LIN {X 0,Y 418.316,Z 278.186,A -85,B 0,C 180,E1 -10001.631,E2 -10001.631} C_VEL
LIN {X 0,Y 418.304,Z 278.193,A -85,B 0,C 180,E1 -10004.596,E2 -10004.596} C_VEL
LIN {X 0,Y 418.281,Z 278.19,A -85,B 0,C 180,E1 -10007.604,E2 -10007.604} C_VEL
LIN {X 0,Y 418.25,Z 278.202,A -85,B 0,C 180,E1 -10010.662,E2 -10010.662} C_VEL
LIN {X 0,Y 418.276,Z 278.19,A -85,B 0,C 180,E1 -10013.781,E2 -10013.781} C_VEL
LIN {X 0,Y 418.309,Z 278.192,A -85,B 0,C 180,E1 -10017.07,E2 -10017.07} C_VEL
LIN {X 0,Y 418.242,Z 278.195,A -85,B 0,C 180,E1 -10020.271,E2 -10020.271} C_VEL
LIN {X 0,Y 418.244,Z 278.196,A -85,B 0,C 180,E1 -10023.676,E2 -10023.676} C_VEL
LIN {X 0,Y 418.236,Z 278.204,A -85,B 0,C 180,E1 -10027.223,E2 -10027.223} C_VEL
LIN {X 0,Y 418.247,Z 278.197,A -85,B 0,C 180,E1 -10029.681,E2 -10029.681} C_VEL
LIN {X 0,Y 418.224,Z 278.197,A -85,B 0,C 180,E1 -10032.32,E2 -10032.32} C_VEL
LIN {X 0,Y 418.253,Z 278.196,A -85,B 0,C 180,E1 -10035.111,E2 -10035.111} C_VEL
LIN {X 0,Y 418.286,Z 278.195,A -85,B 0,C 180,E1 -10037.772,E2 -10037.772} C_VEL
LIN {X 0,Y 418.258,Z 278.198,A -85,B 0,C 180,E1 -10041.559,E2 -10041.559} C_VEL
LIN {X 0,Y 418.252,Z 278.194,A -85,B 0,C 180,E1 -10045.158,E2 -10045.158} C_VEL
LIN {X 0,Y 418.237,Z 278.197,A -85,B 0,C 180,E1 -10047.471,E2 -10047.471} C_VEL
LIN {X 0,Y 418.268,Z 278.192,A -85,B 0,C 180,E1 -10050.893,E2 -10050.893} C_VEL
LIN {X 0,Y 418.262,Z 278.199,A -85,B 0,C 180,E1 -10054.095,E2 -10054.095} C_VEL
LIN {X 0,Y 418.228,Z 278.196,A -85,B 0,C 180,E1 -10057.263,E2 -10057.263} C_VEL
LIN {X 0,Y 418.272,Z 278.198,A -85,B 0,C 180,E1 -10060.364,E2 -10060.364} C_VEL
LIN {X 0,Y 418.306,Z 278.187,A -85,B 0,C 180,E1 -10063.404,E2 -10063.404} C_VEL
LIN {X 0,Y 418.335,Z 278.186,A -85,B 0,C 180,E1 -10066.999,E2 -10066.999} C_VEL
LIN {X 0,Y 418.329,Z 278.186,A -85,B 0,C 180,E1 -10070.328,E2 -10070.328} C_VEL
LIN {X 0,Y 418.479,Z 278.168,A -85,B 0,C 180,E1 -10073.249,E2 -10073.249} C_VEL
LIN {X 0,Y 418.326,Z 278.189,A -85,B 0,C 180,E1 -10075.181,E2 -10075.181} C_VEL
LIN {X 0,Y 418.532,Z 278.158,A -85,B 0,C 180,E1 -10078.075,E2 -10078.075} C_VEL
LIN {X 0,Y 418.659,Z 278.143,A -85,B 0,C 180,E1 -10080,E2 -10080} C_VEL
LIN {X 0,Y 418.489,Z 278.168,A -85,B 0,C 180,E1 -10082.888,E2 -10082.888} C_VEL
LIN {X 0,Y 418.478,Z 278.166,A -85,B 0,C 180,E1 -10086.751,E2 -10086.751} C_VEL
LIN {X 0,Y 418.333,Z 278.188,A -85,B 0,C 180,E1 -10089.671,E2 -10089.671} C_VEL
LIN {X 0,Y 418.344,Z 278.183,A -85,B 0,C 180,E1 -10093.006,E2 -10093.006} C_VEL
LIN {X 0,Y 418.301,Z 278.187,A -85,B 0,C 180,E1 -10096.736,E2 -10096.736} C_VEL
LIN {X 0,Y 418.259,Z 278.201,A -85,B 0,C 180,E1 -10099.79,E2 -10099.79} C_VEL
LIN {X 0,Y 418.221,Z 278.197,A -85,B 0,C 180,E1 -10102.737,E2 -10102.737} C_VEL
LIN {X 0,Y 418.26,Z 278.199,A -85,B 0,C 180,E1 -10105.905,E2 -10105.905} C_VEL
LIN {X 0,Y 418.255,Z 278.193,A -85,B 0,C 180,E1 -10109.163,E2 -10109.163} C_VEL
LIN {X 0,Y 418.248,Z 278.195,A -85,B 0,C 180,E1 -10112.844,E2 -10112.844} C_VEL
LIN {X 0,Y 418.236,Z 278.201,A -85,B 0,C 180,E1 -10116.239,E2 -10116.239} C_VEL
LIN {X 0,Y 418.234,Z 278.196,A -85,B 0,C 180,E1 -10119.684,E2 -10119.684} C_VEL
LIN {X 0,Y 418.221,Z 278.201,A -85,B 0,C 180,E1 -10122.322,E2 -10122.322} C_VEL
LIN {X 0,Y 418.228,Z 278.199,A -85,B 0,C 180,E1 -10125.109,E2 -10125.109} C_VEL
LIN {X 0,Y 418.227,Z 278.196,A -85,B 0,C 180,E1 -10127.767,E2 -10127.767} C_VEL
LIN {X 0,Y 418.239,Z 278.199,A -85,B 0,C 180,E1 -10130.622,E2 -10130.622} C_VEL
LIN {X 0,Y 418.237,Z 278.195,A -85,B 0,C 180,E1 -10133.976,E2 -10133.976} C_VEL
LIN {X 0,Y 418.253,Z 278.201,A -85,B 0,C 180,E1 -10137.157,E2 -10137.157} C_VEL
LIN {X 0,Y 418.257,Z 278.195,A -85,B 0,C 180,E1 -10140.838,E2 -10140.838} C_VEL
LIN {X 0,Y 418.232,Z 278.2,A -85,B 0,C 180,E1 -10144.094,E2 -10144.094} C_VEL
LIN {X 0,Y 418.297,Z 278.248,A -85,B 0,C 180,E1 -10145.383,E2 -10145.383} C_VEL
LIN {X 0,Y 419.802,Z 287.198,A -85,B 0,C 180,E1 -10147.614,E2 -10147.614} C_VEL
LIN {X 0,Y 419.566,Z 294.798,A -85,B 0,C 180,E1 -10149.405,E2 -10149.405} C_VEL
LIN {X 0,Y 418.73,Z 310.631,A -85,B 0,C 180,E1 -10153.076,E2 -10153.076} C_VEL
LIN {X 0,Y 418.286,Z 319.656,A -85,B 0,C 180,E1 -10155.107,E2 -10155.107} C_VEL
LIN {X 0,Y 421.063,Z 340.825,A -85,B 0,C 180,E1 -10155.575,E2 -10155.575} C_VEL
LIN {X 0,Y 420.575,Z 396.454,A -85,B 0,C 180,E1 -10156.563,E2 -10156.563} C_VEL
LIN {X 0,Y 420.25,Z 406.211,A -85,B 0,C 180,E1 -10156.86,E2 -10156.86} C_VEL
LIN {X 0,Y 419.815,Z 417.318,A -85,B 0,C 180,E1 -10157.369,E2 -10157.369} C_VEL
LIN {X 0,Y 419.369,Z 427.432,A -85,B 0,C 180,E1 -10158.031,E2 -10158.031} C_VEL
LIN {X 0,Y 418.942,Z 435.998,A -85,B 0,C 180,E1 -10158.755,E2 -10158.755} C_VEL
LIN {X 0,Y 418.522,Z 444.065,A -85,B 0,C 180,E1 -10159.6,E2 -10159.6} C_VEL
LIN {X 0,Y 418.187,Z 449.871,A -85,B 0,C 180,E1 -10160.325,E2 -10160.325} C_VEL
LIN {X 0,Y 417.792,Z 456.339,A -85,B 0,C 180,E1 -10161.292,E2 -10161.292} C_VEL
LIN {X 0,Y 417.519,Z 461.715,A -85,B 0,C 180,E1 -10162.261,E2 -10162.261} C_VEL
LIN {X 0,Y 417.371,Z 466.202,A -85,B 0,C 180,E1 -10163.231,E2 -10163.231} C_VEL
LIN {X 0,Y 417.197,Z 469.936,A -85,B 0,C 180,E1 -10164.199,E2 -10164.199} C_VEL
LIN {X 0,Y 417.167,Z 472.977,A -85,B 0,C 180,E1 -10165.168,E2 -10165.168} C_VEL
LIN {X 0,Y 417.041,Z 475.336,A -85,B 0,C 180,E1 -10166.135,E2 -10166.135} C_VEL
LIN {X 0,Y 417.041,Z 477.142,A -85,B 0,C 180,E1 -10167.102,E2 -10167.102} C_VEL
LIN {X 0,Y 417.056,Z 478.443,A -85,B 0,C 180,E1 -10168.069,E2 -10168.069} C_VEL
LIN {X 0,Y 417.008,Z 479.263,A -85,B 0,C 180,E1 -10169.034,E2 -10169.034} C_VEL
LIN {X 0,Y 417.002,Z 479.568,A -85,B 0,C 180,E1 -10170,E2 -10170} C_VEL
LIN {X 0,Y 417.008,Z 479.285,A -85,B 0,C 180,E1 -10170.966,E2 -10170.966} C_VEL
LIN {X 0,Y 417.056,Z 478.529,A -85,B 0,C 180,E1 -10171.931,E2 -10171.931} C_VEL
LIN {X 0,Y 417.04,Z 477.294,A -85,B 0,C 180,E1 -10172.898,E2 -10172.898} C_VEL
LIN {X 0,Y 417.088,Z 474.395,A -85,B 0,C 180,E1 -10174.349,E2 -10174.349} C_VEL
LIN {X 0,Y 417.192,Z 471.764,A -85,B 0,C 180,E1 -10175.316,E2 -10175.316} C_VEL
LIN {X 0,Y 417.322,Z 467.715,A -85,B 0,C 180,E1 -10176.486,E2 -10176.486} C_VEL
LIN {X 0,Y 417.538,Z 462.205,A -85,B 0,C 180,E1 -10177.738,E2 -10177.738} C_VEL
LIN {X 0,Y 417.8,Z 456.96,A -85,B 0,C 180,E1 -10178.707,E2 -10178.707} C_VEL
LIN {X 0,Y 418.226,Z 450.654,A -85,B 0,C 180,E1 -10179.674,E2 -10179.674} C_VEL
LIN {X 0,Y 418.713,Z 442.99,A -85,B 0,C 180,E1 -10180.639,E2 -10180.639} C_VEL
LIN {X 0,Y 419.187,Z 433.445,A -85,B 0,C 180,E1 -10181.606,E2 -10181.606} C_VEL
LIN {X 0,Y 419.711,Z 424.117,A -85,B 0,C 180,E1 -10182.327,E2 -10182.327} C_VEL
LIN {X 0,Y 420.105,Z 415.129,A -85,B 0,C 180,E1 -10182.868,E2 -10182.868} C_VEL
LIN {X 0,Y 420.483,Z 405.772,A -85,B 0,C 180,E1 -10183.286,E2 -10183.286} C_VEL
LIN {X 0,Y 420.789,Z 397.063,A -85,B 0,C 180,E1 -10183.556,E2 -10183.556} C_VEL
LIN {X 0,Y 421.222,Z 353.269,A -85,B 0,C 180,E1 -10184.347,E2 -10184.347} C_VEL
LIN {X 0,Y 421.201,Z 339.749,A -85,B 0,C 180,E1 -10184.588,E2 -10184.588} C_VEL
LIN {X 0,Y 418.296,Z 318.919,A -85,B 0,C 180,E1 -10185.079,E2 -10185.079} C_VEL
LIN {X 0,Y 419.059,Z 303.357,A -85,B 0,C 180,E1 -10188.581,E2 -10188.581} C_VEL
LIN {X 0,Y 419.807,Z 288.926,A -85,B 0,C 180,E1 -10191.868,E2 -10191.868} C_VEL
LIN {X 0,Y 419.482,Z 284.742,A -85,B 0,C 180,E1 -10192.858,E2 -10192.858} C_VEL
LIN {X 0,Y 418.312,Z 278.194,A -85,B 0,C 180,E1 -10194.504,E2 -10194.504} C_VEL
LIN {X 0,Y 418.213,Z 278.204,A -85,B 0,C 180,E1 -10198.068,E2 -10198.068} C_VEL
LIN {X 0,Y 418.206,Z 278.202,A -85,B 0,C 180,E1 -10201.395,E2 -10201.395} C_VEL
LIN {X 0,Y 418.259,Z 278.198,A -85,B 0,C 180,E1 -10204.579,E2 -10204.579} C_VEL
LIN {X 0,Y 418.22,Z 278.203,A -85,B 0,C 180,E1 -10207.832,E2 -10207.832} C_VEL
LIN {X 0,Y 418.213,Z 278.209,A -85,B 0,C 180,E1 -10210.948,E2 -10210.948} C_VEL
LIN {X 0,Y 418.201,Z 278.207,A -85,B 0,C 180,E1 -10213.728,E2 -10213.728} C_VEL
LIN {X 0,Y 418.201,Z 278.203,A -85,B 0,C 180,E1 -10216.448,E2 -10216.448} C_VEL
LIN {X 0,Y 418.215,Z 278.201,A -85,B 0,C 180,E1 -10219.129,E2 -10219.129} C_VEL
LIN {X 0,Y 418.216,Z 278.196,A -85,B 0,C 180,E1 -10222.166,E2 -10222.166} C_VEL
LIN {X 0,Y 418.256,Z 278.198,A -85,B 0,C 180,E1 -10225.419,E2 -10225.419} C_VEL
LIN {X 0,Y 418.201,Z 278.199,A -85,B 0,C 180,E1 -10228.603,E2 -10228.603} C_VEL
LIN {X 0,Y 418.28,Z 278.19,A -85,B 0,C 180,E1 -10231.936,E2 -10231.936} C_VEL
LIN {X 0,Y 418.279,Z 278.19,A -85,B 0,C 180,E1 -10235.162,E2 -10235.162} C_VEL
LIN {X 0,Y 418.222,Z 278.195,A -85,B 0,C 180,E1 -10238.303,E2 -10238.303} C_VEL
LIN {X 0,Y 418.271,Z 278.192,A -85,B 0,C 180,E1 -10241.383,E2 -10241.383} C_VEL
LIN {X 0,Y 418.289,Z 278.187,A -85,B 0,C 180,E1 -10244.406,E2 -10244.406} C_VEL
LIN {X 0,Y 418.343,Z 278.183,A -85,B 0,C 180,E1 -10247.385,E2 -10247.385} C_VEL
LIN {X 0,Y 418.329,Z 278.182,A -85,B 0,C 180,E1 -10250.328,E2 -10250.328} C_VEL
LIN {X 0,Y 418.479,Z 278.166,A -85,B 0,C 180,E1 -10253.249,E2 -10253.249} C_VEL
LIN {X 0,Y 418.325,Z 278.182,A -85,B 0,C 180,E1 -10255.181,E2 -10255.181} C_VEL
LIN {X 0,Y 418.528,Z 278.155,A -85,B 0,C 180,E1 -10258.076,E2 -10258.076} C_VEL
LIN {X 0,Y 418.658,Z 278.142,A -85,B 0,C 180,E1 -10260,E2 -10260} C_VEL
LIN {X 0,Y 418.488,Z 278.162,A -85,B 0,C 180,E1 -10262.888,E2 -10262.888} C_VEL
LIN {X 0,Y 418.445,Z 278.17,A -85,B 0,C 180,E1 -10266.51,E2 -10266.51} C_VEL
LIN {X 0,Y 418.329,Z 278.188,A -85,B 0,C 180,E1 -10269.672,E2 -10269.672} C_VEL
LIN {X 0,Y 418.334,Z 278.181,A -85,B 0,C 180,E1 -10273.001,E2 -10273.001} C_VEL
LIN {X 0,Y 418.301,Z 278.185,A -85,B 0,C 180,E1 -10276.736,E2 -10276.736} C_VEL
LIN {X 0,Y 418.259,Z 278.198,A -85,B 0,C 180,E1 -10279.791,E2 -10279.791} C_VEL
LIN {X 0,Y 418.228,Z 278.2,A -85,B 0,C 180,E1 -10282.737,E2 -10282.737} C_VEL
LIN {X 0,Y 418.261,Z 278.199,A -85,B 0,C 180,E1 -10285.905,E2 -10285.905} C_VEL
LIN {X 0,Y 418.265,Z 278.192,A -85,B 0,C 180,E1 -10289.162,E2 -10289.162} C_VEL
LIN {X 0,Y 418.249,Z 278.197,A -85,B 0,C 180,E1 -10292.845,E2 -10292.845} C_VEL
LIN {X 0,Y 418.241,Z 278.203,A -85,B 0,C 180,E1 -10296.24,E2 -10296.24} C_VEL
LIN {X 0,Y 418.258,Z 278.197,A -85,B 0,C 180,E1 -10299.681,E2 -10299.681} C_VEL
LIN {X 0,Y 418.369,Z 278.298,A -85,B 0,C 180,E1 -10302.411,E2 -10302.411} C_VEL
LIN {X 0,Y 418.975,Z 282.45,A -85,B 0,C 180,E1 -10303.452,E2 -10303.452} C_VEL
LIN {X 0,Y 418.645,Z 295.196,A -85,B 0,C 180,E1 -10306.507,E2 -10306.507} C_VEL
LIN {X 0,Y 418.562,Z 297.209,A -85,B 0,C 180,E1 -10306.988,E2 -10306.988} C_VEL
LIN {X 0,Y 421.569,Z 313.989,A -85,B 0,C 180,E1 -10307.407,E2 -10307.407} C_VEL
LIN {X 0,Y 420.868,Z 374.296,A -85,B 0,C 180,E1 -10308.481,E2 -10308.481} C_VEL
LIN {X 0,Y 420.649,Z 384.823,A -85,B 0,C 180,E1 -10308.818,E2 -10308.818} C_VEL
LIN {X 0,Y 420.3,Z 396.213,A -85,B 0,C 180,E1 -10309.378,E2 -10309.378} C_VEL
LIN {X 0,Y 419.835,Z 405.763,A -85,B 0,C 180,E1 -10310.032,E2 -10310.032} C_VEL
LIN {X 0,Y 419.413,Z 414.156,A -85,B 0,C 180,E1 -10310.762,E2 -10310.762} C_VEL
LIN {X 0,Y 419.027,Z 421.038,A -85,B 0,C 180,E1 -10311.49,E2 -10311.49} C_VEL
LIN {X 0,Y 418.58,Z 427.446,A -85,B 0,C 180,E1 -10312.299,E2 -10312.299} C_VEL
LIN {X 0,Y 418.219,Z 434.203,A -85,B 0,C 180,E1 -10313.338,E2 -10313.338} C_VEL
LIN {X 0,Y 417.908,Z 439.094,A -85,B 0,C 180,E1 -10314.241,E2 -10314.241} C_VEL
LIN {X 0,Y 417.688,Z 443.08,A -85,B 0,C 180,E1 -10315.106,E2 -10315.106} C_VEL
LIN {X 0,Y 417.385,Z 447.361,A -85,B 0,C 180,E1 -10316.245,E2 -10316.245} C_VEL
LIN {X 0,Y 417.277,Z 450.729,A -85,B 0,C 180,E1 -10317.388,E2 -10317.388} C_VEL
LIN {X 0,Y 417.158,Z 453.255,A -85,B 0,C 180,E1 -10318.517,E2 -10318.517} C_VEL
LIN {X 0,Y 417.042,Z 455.033,A -85,B 0,C 180,E1 -10319.633,E2 -10319.633} C_VEL
LIN {X 0,Y 416.896,Z 456.103,A -85,B 0,C 180,E1 -10320.734,E2 -10320.734} C_VEL
LIN {X 0,Y 416.833,Z 456.488,A -85,B 0,C 180,E1 -10321.831,E2 -10321.831} C_VEL
LIN {X 0,Y 416.873,Z 456.019,A -85,B 0,C 180,E1 -10323.319,E2 -10323.319} C_VEL
LIN {X 0,Y 417.005,Z 453.825,A -85,B 0,C 180,E1 -10325.082,E2 -10325.082} C_VEL
LIN {X 0,Y 417.242,Z 450.406,A -85,B 0,C 180,E1 -10326.683,E2 -10326.683} C_VEL
LIN {X 0,Y 417.489,Z 445.322,A -85,B 0,C 180,E1 -10328.264,E2 -10328.264} C_VEL
LIN {X 0,Y 417.68,Z 440.977,A -85,B 0,C 180,E1 -10329.308,E2 -10329.308} C_VEL
LIN {X 0,Y 418.017,Z 435.649,A -85,B 0,C 180,E1 -10330.352,E2 -10330.352} C_VEL
LIN {X 0,Y 418.381,Z 429.177,A -85,B 0,C 180,E1 -10331.388,E2 -10331.388} C_VEL
LIN {X 0,Y 418.751,Z 422.34,A -85,B 0,C 180,E1 -10332.291,E2 -10332.291} C_VEL
LIN {X 0,Y 419.202,Z 414.497,A -85,B 0,C 180,E1 -10333.14,E2 -10333.14} C_VEL
LIN {X 0,Y 419.603,Z 406.643,A -85,B 0,C 180,E1 -10333.833,E2 -10333.833} C_VEL
LIN {X 0,Y 420.009,Z 397.564,A -85,B 0,C 180,E1 -10334.471,E2 -10334.471} C_VEL
LIN {X 0,Y 420.305,Z 386.898,A -85,B 0,C 180,E1 -10335.041,E2 -10335.041} C_VEL
LIN {X 0,Y 420.639,Z 375.759,A -85,B 0,C 180,E1 -10335.425,E2 -10335.425} C_VEL
LIN {X 0,Y 420.873,Z 354.388,A -85,B 0,C 180,E1 -10335.832,E2 -10335.832} C_VEL
LIN {X 0,Y 421.091,Z 312.94,A -85,B 0,C 180,E1 -10336.555,E2 -10336.555} C_VEL
LIN {X 0,Y 419.805,Z 308.946,A -85,B 0,C 180,E1 -10336.67,E2 -10336.67} C_VEL
LIN {X 0,Y 416.141,Z 303,A -85,B 0,C 180,E1 -10336.901,E2 -10336.901} C_VEL
LIN {X 0,Y 413.111,Z 298.98,A -85,B 0,C 180,E1 -10337.184,E2 -10337.184} C_VEL
LIN {X 0,Y 411.741,Z 296.621,A -85,B 0,C 180,E1 -10337.5,E2 -10337.5} C_VEL
LIN {X 0,Y 411.55,Z 295.765,A -85,B 0,C 180,E1 -10337.686,E2 -10337.686} C_VEL
LIN {X 0,Y 411.925,Z 284.68,A -85,B 0,C 180,E1 -10340.673,E2 -10340.673} C_VEL
LIN {X 0,Y 411.466,Z 279.045,A -85,B 0,C 180,E1 -10342.277,E2 -10342.277} C_VEL
LIN {X 0,Y 411.473,Z 279.044,A -85,B 0,C 180,E1 -10344.118,E2 -10344.118} C_VEL
LIN {X 0,Y 411.513,Z 279.038,A -85,B 0,C 180,E1 -10348.043,E2 -10348.043} C_VEL
LIN {X 0,Y 411.642,Z 279.024,A -85,B 0,C 180,E1 -10350,E2 -10350} C_VEL
LIN {X 0,Y 411.46,Z 279.039,A -85,B 0,C 180,E1 -10352.937,E2 -10352.937} C_VEL
LIN {X 0,Y 411.46,Z 279.044,A -85,B 0,C 180,E1 -10355.882,E2 -10355.882} C_VEL
LIN {X 0,Y 411.353,Z 279.054,A -85,B 0,C 180,E1 -10358.845,E2 -10358.845} C_VEL
LIN {X 0,Y 411.284,Z 279.063,A -85,B 0,C 180,E1 -10361.832,E2 -10361.832} C_VEL
LIN {X 0,Y 411.261,Z 279.067,A -85,B 0,C 180,E1 -10364.852,E2 -10364.852} C_VEL
LIN {X 0,Y 411.246,Z 279.067,A -85,B 0,C 180,E1 -10367.915,E2 -10367.915} C_VEL
LIN {X 0,Y 411.196,Z 279.075,A -85,B 0,C 180,E1 -10371.033,E2 -10371.033} C_VEL
LIN {X 0,Y 411.219,Z 279.071,A -85,B 0,C 180,E1 -10374.215,E2 -10374.215} C_VEL
LIN {X 0,Y 411.258,Z 279.066,A -85,B 0,C 180,E1 -10377.477,E2 -10377.477} C_VEL
LIN {X 0,Y 411.187,Z 279.079,A -85,B 0,C 180,E1 -10380.847,E2 -10380.847} C_VEL
LIN {X 0,Y 411.201,Z 279.072,A -85,B 0,C 180,E1 -10384.333,E2 -10384.333} C_VEL
LIN {X 0,Y 411.191,Z 279.073,A -85,B 0,C 180,E1 -10387.973,E2 -10387.973} C_VEL
LIN {X 0,Y 411.177,Z 279.075,A -85,B 0,C 180,E1 -10390.503,E2 -10390.503} C_VEL
LIN {X 0,Y 411.168,Z 279.08,A -85,B 0,C 180,E1 -10393.133,E2 -10393.133} C_VEL
LIN {X 0,Y 411.222,Z 279.073,A -85,B 0,C 180,E1 -10395.872,E2 -10395.872} C_VEL
LIN {X 0,Y 411.203,Z 279.071,A -85,B 0,C 180,E1 -10398.763,E2 -10398.763} C_VEL
LIN {X 0,Y 411.197,Z 279.077,A -85,B 0,C 180,E1 -10402.026,E2 -10402.026} C_VEL
LIN {X 0,Y 411.199,Z 279.077,A -85,B 0,C 180,E1 -10405.666,E2 -10405.666} C_VEL
LIN {X 0,Y 411.189,Z 279.073,A -85,B 0,C 180,E1 -10409.152,E2 -10409.152} C_VEL
LIN {X 0,Y 411.251,Z 279.068,A -85,B 0,C 180,E1 -10412.522,E2 -10412.522} C_VEL
LIN {X 0,Y 411.217,Z 279.072,A -85,B 0,C 180,E1 -10415.784,E2 -10415.784} C_VEL
LIN {X 0,Y 411.186,Z 279.075,A -85,B 0,C 180,E1 -10418.965,E2 -10418.965} C_VEL
LIN {X 0,Y 411.241,Z 279.07,A -85,B 0,C 180,E1 -10422.084,E2 -10422.084} C_VEL
LIN {X 0,Y 411.249,Z 279.067,A -85,B 0,C 180,E1 -10425.147,E2 -10425.147} C_VEL
LIN {X 0,Y 411.272,Z 279.065,A -85,B 0,C 180,E1 -10428.167,E2 -10428.167} C_VEL
LIN {X 0,Y 411.432,Z 279.044,A -85,B 0,C 180,E1 -10432.186,E2 -10432.186} C_VEL
LIN {X 0,Y 411.459,Z 279.04,A -85,B 0,C 180,E1 -10434.118,E2 -10434.118} C_VEL
LIN {X 0,Y 411.502,Z 279.034,A -85,B 0,C 180,E1 -10438.042,E2 -10438.042} C_VEL
LIN {X 0,Y 411.629,Z 279.018,A -85,B 0,C 180,E1 -10440,E2 -10440} C_VEL
LIN {X 0,Y 411.446,Z 279.046,A -85,B 0,C 180,E1 -10442.937,E2 -10442.937} C_VEL
LIN {X 0,Y 411.442,Z 279.044,A -85,B 0,C 180,E1 -10446.867,E2 -10446.867} C_VEL
LIN {X 0,Y 411.286,Z 279.064,A -85,B 0,C 180,E1 -10449.839,E2 -10449.839} C_VEL
LIN {X 0,Y 411.302,Z 279.061,A -85,B 0,C 180,E1 -10453.109,E2 -10453.109} C_VEL
LIN {X 0,Y 411.246,Z 279.066,A -85,B 0,C 180,E1 -10456.889,E2 -10456.889} C_VEL
LIN {X 0,Y 411.22,Z 279.075,A -85,B 0,C 180,E1 -10459.987,E2 -10459.987} C_VEL
LIN {X 0,Y 411.186,Z 279.074,A -85,B 0,C 180,E1 -10463.148,E2 -10463.148} C_VEL
LIN {X 0,Y 411.228,Z 279.072,A -85,B 0,C 180,E1 -10466.381,E2 -10466.381} C_VEL
LIN {X 0,Y 411.19,Z 279.076,A -85,B 0,C 180,E1 -10469.713,E2 -10469.713} C_VEL
LIN {X 0,Y 411.197,Z 279.072,A -85,B 0,C 180,E1 -10473.156,E2 -10473.156} C_VEL
LIN {X 0,Y 411.184,Z 279.08,A -85,B 0,C 180,E1 -10476.553,E2 -10476.553} C_VEL
LIN {X 0,Y 411.199,Z 279.072,A -85,B 0,C 180,E1 -10479.728,E2 -10479.728} C_VEL
LIN {X 0,Y 411.165,Z 279.078,A -85,B 0,C 180,E1 -10483.135,E2 -10483.135} C_VEL
LIN {X 0,Y 411.16,Z 279.077,A -85,B 0,C 180,E1 -10485.882,E2 -10485.882} C_VEL
LIN {X 0,Y 411.154,Z 279.085,A -85,B 0,C 180,E1 -10488.773,E2 -10488.773} C_VEL
LIN {X 0,Y 411.186,Z 279.073,A -85,B 0,C 180,E1 -10492.027,E2 -10492.027} C_VEL
LIN {X 0,Y 411.2,Z 279.073,A -85,B 0,C 180,E1 -10495.667,E2 -10495.667} C_VEL
LIN {X 0,Y 411.185,Z 279.081,A -85,B 0,C 180,E1 -10499.153,E2 -10499.153} C_VEL
LIN {X 0,Y 411.184,Z 279.077,A -85,B 0,C 180,E1 -10502.518,E2 -10502.518} C_VEL
LIN {X 0,Y 411.27,Z 279.187,A -85,B 0,C 180,E1 -10505.229,E2 -10505.229} C_VEL
LIN {X 0,Y 412.803,Z 288.036,A -85,B 0,C 180,E1 -10507.477,E2 -10507.477} C_VEL
LIN {X 0,Y 412.655,Z 294.551,A -85,B 0,C 180,E1 -10509.044,E2 -10509.044} C_VEL
LIN {X 0,Y 411.717,Z 311,A -85,B 0,C 180,E1 -10512.924,E2 -10512.924} C_VEL
LIN {X 0,Y 411.263,Z 319.493,A -85,B 0,C 180,E1 -10514.863,E2 -10514.863} C_VEL
LIN {X 0,Y 414.18,Z 341.57,A -85,B 0,C 180,E1 -10515.363,E2 -10515.363} C_VEL
LIN {X 0,Y 413.656,Z 396.845,A -85,B 0,C 180,E1 -10516.365,E2 -10516.365} C_VEL
LIN {X 0,Y 413.242,Z 408.043,A -85,B 0,C 180,E1 -10516.727,E2 -10516.727} C_VEL
LIN {X 0,Y 412.768,Z 419.816,A -85,B 0,C 180,E1 -10517.337,E2 -10517.337} C_VEL
LIN {X 0,Y 412.32,Z 428.534,A -85,B 0,C 180,E1 -10517.948,E2 -10517.948} C_VEL
LIN {X 0,Y 411.908,Z 436.868,A -85,B 0,C 180,E1 -10518.685,E2 -10518.685} C_VEL
LIN {X 0,Y 411.454,Z 444.755,A -85,B 0,C 180,E1 -10519.544,E2 -10519.544} C_VEL
LIN {X 0,Y 411.056,Z 451.273,A -85,B 0,C 180,E1 -10520.404,E2 -10520.404} C_VEL
LIN {X 0,Y 410.678,Z 457.476,A -85,B 0,C 180,E1 -10521.388,E2 -10521.388} C_VEL
LIN {X 0,Y 410.405,Z 462.624,A -85,B 0,C 180,E1 -10522.374,E2 -10522.374} C_VEL
LIN {X 0,Y 410.328,Z 465.947,A -85,B 0,C 180,E1 -10523.114,E2 -10523.114} C_VEL
LIN {X 0,Y 410.112,Z 469.693,A -85,B 0,C 180,E1 -10524.099,E2 -10524.099} C_VEL
LIN {X 0,Y 410.079,Z 472.741,A -85,B 0,C 180,E1 -10525.084,E2 -10525.084} C_VEL
LIN {X 0,Y 409.959,Z 475.108,A -85,B 0,C 180,E1 -10526.068,E2 -10526.068} C_VEL
LIN {X 0,Y 409.939,Z 476.923,A -85,B 0,C 180,E1 -10527.052,E2 -10527.052} C_VEL
LIN {X 0,Y 409.967,Z 478.234,A -85,B 0,C 180,E1 -10528.035,E2 -10528.035} C_VEL
LIN {X 0,Y 409.933,Z 479.063,A -85,B 0,C 180,E1 -10529.018,E2 -10529.018} C_VEL
LIN {X 0,Y 409.924,Z 479.369,A -85,B 0,C 180,E1 -10530,E2 -10530} C_VEL
LIN {X 0,Y 409.933,Z 479.093,A -85,B 0,C 180,E1 -10530.982,E2 -10530.982} C_VEL
LIN {X 0,Y 409.967,Z 478.345,A -85,B 0,C 180,E1 -10531.965,E2 -10531.965} C_VEL
LIN {X 0,Y 409.938,Z 477.118,A -85,B 0,C 180,E1 -10532.948,E2 -10532.948} C_VEL
LIN {X 0,Y 410.019,Z 474.229,A -85,B 0,C 180,E1 -10534.424,E2 -10534.424} C_VEL
LIN {X 0,Y 410.111,Z 471.606,A -85,B 0,C 180,E1 -10535.408,E2 -10535.408} C_VEL
LIN {X 0,Y 410.327,Z 466.438,A -85,B 0,C 180,E1 -10536.886,E2 -10536.886} C_VEL
LIN {X 0,Y 410.545,Z 460.884,A -85,B 0,C 180,E1 -10538.119,E2 -10538.119} C_VEL
LIN {X 0,Y 411.011,Z 453.936,A -85,B 0,C 180,E1 -10539.348,E2 -10539.348} C_VEL
LIN {X 0,Y 411.547,Z 445.969,A -85,B 0,C 180,E1 -10540.453,E2 -10540.453} C_VEL
LIN {X 0,Y 411.957,Z 438.37,A -85,B 0,C 180,E1 -10541.314,E2 -10541.314} C_VEL
LIN {X 0,Y 412.434,Z 430.419,A -85,B 0,C 180,E1 -10542.048,E2 -10542.048} C_VEL
LIN {X 0,Y 412.86,Z 422.231,A -85,B 0,C 180,E1 -10542.66,E2 -10542.66} C_VEL
LIN {X 0,Y 413.246,Z 413.963,A -85,B 0,C 180,E1 -10543.147,E2 -10543.147} C_VEL
LIN {X 0,Y 413.625,Z 405.078,A -85,B 0,C 180,E1 -10543.542,E2 -10543.542} C_VEL
LIN {X 0,Y 413.961,Z 396.013,A -85,B 0,C 180,E1 -10543.817,E2 -10543.817} C_VEL
LIN {X 0,Y 414.394,Z 340.622,A -85,B 0,C 180,E1 -10544.827,E2 -10544.827} C_VEL
LIN {X 0,Y 411.319,Z 318.63,A -85,B 0,C 180,E1 -10545.376,E2 -10545.376} C_VEL
LIN {X 0,Y 412.108,Z 303.217,A -85,B 0,C 180,E1 -10548.906,E2 -10548.906} C_VEL
LIN {X 0,Y 412.884,Z 288.776,A -85,B 0,C 180,E1 -10552.254,E2 -10552.254} C_VEL
LIN {X 0,Y 411.245,Z 279.074,A -85,B 0,C 180,E1 -10554.709,E2 -10554.709} C_VEL
LIN {X 0,Y 411.174,Z 279.083,A -85,B 0,C 180,E1 -10558.592,E2 -10558.592} C_VEL
LIN {X 0,Y 411.161,Z 279.078,A -85,B 0,C 180,E1 -10561.997,E2 -10561.997} C_VEL
LIN {X 0,Y 411.205,Z 279.078,A -85,B 0,C 180,E1 -10564.877,E2 -10564.877} C_VEL
LIN {X 0,Y 411.196,Z 279.078,A -85,B 0,C 180,E1 -10568.167,E2 -10568.167} C_VEL
LIN {X 0,Y 411.154,Z 279.087,A -85,B 0,C 180,E1 -10571.227,E2 -10571.227} C_VEL
LIN {X 0,Y 411.168,Z 279.081,A -85,B 0,C 180,E1 -10574.49,E2 -10574.49} C_VEL
LIN {X 0,Y 411.169,Z 279.076,A -85,B 0,C 180,E1 -10578.194,E2 -10578.194} C_VEL
LIN {X 0,Y 411.2,Z 279.074,A -85,B 0,C 180,E1 -10580.774,E2 -10580.774} C_VEL
LIN {X 0,Y 411.189,Z 279.074,A -85,B 0,C 180,E1 -10584.47,E2 -10584.47} C_VEL
LIN {X 0,Y 411.198,Z 279.07,A -85,B 0,C 180,E1 -10586.873,E2 -10586.873} C_VEL
LIN {X 0,Y 411.223,Z 279.069,A -85,B 0,C 180,E1 -10590.644,E2 -10590.644} C_VEL
LIN {X 0,Y 411.226,Z 279.066,A -85,B 0,C 180,E1 -10593.618,E2 -10593.618} C_VEL
LIN {X 0,Y 411.184,Z 279.072,A -85,B 0,C 180,E1 -10596.851,E2 -10596.851} C_VEL
LIN {X 0,Y 411.203,Z 279.073,A -85,B 0,C 180,E1 -10600.05,E2 -10600.05} C_VEL
LIN {X 0,Y 411.252,Z 279.062,A -85,B 0,C 180,E1 -10603.131,E2 -10603.131} C_VEL
LIN {X 0,Y 411.293,Z 279.064,A -85,B 0,C 180,E1 -10606.896,E2 -10606.896} C_VEL
LIN {X 0,Y 411.281,Z 279.061,A -85,B 0,C 180,E1 -10610.161,E2 -10610.161} C_VEL
LIN {X 0,Y 411.446,Z 279.043,A -85,B 0,C 180,E1 -10613.133,E2 -10613.133} C_VEL
LIN {X 0,Y 411.296,Z 279.058,A -85,B 0,C 180,E1 -10615.099,E2 -10615.099} C_VEL
LIN {X 0,Y 411.498,Z 279.031,A -85,B 0,C 180,E1 -10618.043,E2 -10618.043} C_VEL
LIN {X 0,Y 411.628,Z 279.018,A -85,B 0,C 180,E1 -10620,E2 -10620} C_VEL
LIN {X 0,Y 411.445,Z 279.039,A -85,B 0,C 180,E1 -10622.937,E2 -10622.937} C_VEL
LIN {X 0,Y 411.411,Z 279.049,A -85,B 0,C 180,E1 -10626.868,E2 -10626.868} C_VEL
LIN {X 0,Y 411.281,Z 279.065,A -85,B 0,C 180,E1 -10629.839,E2 -10629.839} C_VEL
LIN {X 0,Y 411.294,Z 279.059,A -85,B 0,C 180,E1 -10633.104,E2 -10633.104} C_VEL
LIN {X 0,Y 411.246,Z 279.065,A -85,B 0,C 180,E1 -10636.889,E2 -10636.889} C_VEL
LIN {X 0,Y 411.22,Z 279.073,A -85,B 0,C 180,E1 -10639.987,E2 -10639.987} C_VEL
LIN {X 0,Y 411.193,Z 279.077,A -85,B 0,C 180,E1 -10643.148,E2 -10643.148} C_VEL
LIN {X 0,Y 411.229,Z 279.071,A -85,B 0,C 180,E1 -10646.382,E2 -10646.382} C_VEL
LIN {X 0,Y 411.201,Z 279.076,A -85,B 0,C 180,E1 -10649.713,E2 -10649.713} C_VEL
LIN {X 0,Y 411.198,Z 279.075,A -85,B 0,C 180,E1 -10653.157,E2 -10653.157} C_VEL
LIN {X 0,Y 411.188,Z 279.08,A -85,B 0,C 180,E1 -10656.554,E2 -10656.554} C_VEL
LIN {X 0,Y 411.22,Z 279.075,A -85,B 0,C 180,E1 -10659.731,E2 -10659.731} C_VEL
LIN {X 0,Y 411.31,Z 279.257,A -85,B 0,C 180,E1 -10662.241,E2 -10662.241} C_VEL
LIN {X 0,Y 411.99,Z 283.493,A -85,B 0,C 180,E1 -10663.324,E2 -10663.324} C_VEL
LIN {X 0,Y 411.703,Z 294.473,A -85,B 0,C 180,E1 -10665.999,E2 -10665.999} C_VEL
LIN {X 0,Y 411.613,Z 297.373,A -85,B 0,C 180,E1 -10666.701,E2 -10666.701} C_VEL
LIN {X 0,Y 414.651,Z 313.973,A -85,B 0,C 180,E1 -10667.139,E2 -10667.139} C_VEL
LIN {X 0,Y 414.007,Z 374.628,A -85,B 0,C 180,E1 -10668.243,E2 -10668.243} C_VEL
LIN {X 0,Y 413.748,Z 385.397,A -85,B 0,C 180,E1 -10668.595,E2 -10668.595} C_VEL
LIN {X 0,Y 413.363,Z 397.087,A -85,B 0,C 180,E1 -10669.194,E2 -10669.194} C_VEL
LIN {X 0,Y 412.921,Z 405.873,A -85,B 0,C 180,E1 -10669.807,E2 -10669.807} C_VEL
LIN {X 0,Y 412.532,Z 413.354,A -85,B 0,C 180,E1 -10670.457,E2 -10670.457} C_VEL
LIN {X 0,Y 412.16,Z 419.843,A -85,B 0,C 180,E1 -10671.129,E2 -10671.129} C_VEL
LIN {X 0,Y 411.611,Z 427.326,A -85,B 0,C 180,E1 -10672.073,E2 -10672.073} C_VEL
LIN {X 0,Y 411.31,Z 433.193,A -85,B 0,C 180,E1 -10672.966,E2 -10672.966} C_VEL
LIN {X 0,Y 410.882,Z 439.508,A -85,B 0,C 180,E1 -10674.139,E2 -10674.139} C_VEL
LIN {X 0,Y 410.571,Z 444.353,A -85,B 0,C 180,E1 -10675.25,E2 -10675.25} C_VEL
LIN {X 0,Y 410.253,Z 449.481,A -85,B 0,C 180,E1 -10676.758,E2 -10676.758} C_VEL
LIN {X 0,Y 410.136,Z 452.37,A -85,B 0,C 180,E1 -10677.914,E2 -10677.914} C_VEL
LIN {X 0,Y 410.017,Z 454.457,A -85,B 0,C 180,E1 -10679.056,E2 -10679.056} C_VEL
LIN {X 0,Y 409.869,Z 455.821,A -85,B 0,C 180,E1 -10680.182,E2 -10680.182} C_VEL
LIN {X 0,Y 409.755,Z 456.523,A -85,B 0,C 180,E1 -10681.299,E2 -10681.299} C_VEL
LIN {X 0,Y 409.792,Z 456.354,A -85,B 0,C 180,E1 -10683.102,E2 -10683.102} C_VEL
LIN {X 0,Y 409.867,Z 454.852,A -85,B 0,C 180,E1 -10684.617,E2 -10684.617} C_VEL
LIN {X 0,Y 410.007,Z 453.018,A -85,B 0,C 180,E1 -10685.709,E2 -10685.709} C_VEL
LIN {X 0,Y 410.235,Z 449.087,A -85,B 0,C 180,E1 -10687.276,E2 -10687.276} C_VEL
LIN {X 0,Y 410.5,Z 444.305,A -85,B 0,C 180,E1 -10688.666,E2 -10688.666} C_VEL
LIN {X 0,Y 410.763,Z 439.677,A -85,B 0,C 180,E1 -10689.729,E2 -10689.729} C_VEL
LIN {X 0,Y 411.066,Z 433.98,A -85,B 0,C 180,E1 -10690.801,E2 -10690.801} C_VEL
LIN {X 0,Y 411.488,Z 427.242,A -85,B 0,C 180,E1 -10691.839,E2 -10691.839} C_VEL
LIN {X 0,Y 412.018,Z 418.548,A -85,B 0,C 180,E1 -10692.923,E2 -10692.923} C_VEL
LIN {X 0,Y 412.503,Z 409.493,A -85,B 0,C 180,E1 -10693.801,E2 -10693.801} C_VEL
LIN {X 0,Y 412.915,Z 401.063,A -85,B 0,C 180,E1 -10694.451,E2 -10694.451} C_VEL
LIN {X 0,Y 413.269,Z 391.303,A -85,B 0,C 180,E1 -10695.033,E2 -10695.033} C_VEL
LIN {X 0,Y 413.511,Z 382.229,A -85,B 0,C 180,E1 -10695.432,E2 -10695.432} C_VEL
LIN {X 0,Y 413.749,Z 372.445,A -85,B 0,C 180,E1 -10695.72,E2 -10695.72} C_VEL
LIN {X 0,Y 414.211,Z 313.901,A -85,B 0,C 180,E1 -10696.772,E2 -10696.772} C_VEL
LIN {X 0,Y 411.455,Z 297.696,A -85,B 0,C 180,E1 -10697.171,E2 -10697.171} C_VEL
LIN {X 0,Y 411.55,Z 295.765,A -85,B 0,C 180,E1 -10697.686,E2 -10697.686} C_VEL
LIN {X 0,Y 410.962,Z 293.144,A -85,B 0,C 180,E1 -10698.419,E2 -10698.419} C_VEL
LIN {X 0,Y 405.183,Z 284.338,A -85,B 0,C 180,E1 -10701.112,E2 -10701.112} C_VEL
LIN {X 0,Y 404.788,Z 282.599,A -85,B 0,C 180,E1 -10701.616,E2 -10701.616} C_VEL
LIN {X 0,Y 404.399,Z 279.924,A -85,B 0,C 180,E1 -10702.438,E2 -10702.438} C_VEL
LIN {X 0,Y 404.282,Z 279.934,A -85,B 0,C 180,E1 -10705.014,E2 -10705.014} C_VEL
LIN {X 0,Y 404.482,Z 279.914,A -85,B 0,C 180,E1 -10708.009,E2 -10708.009} C_VEL
LIN {X 0,Y 404.612,Z 279.899,A -85,B 0,C 180,E1 -10710,E2 -10710} C_VEL
LIN {X 0,Y 404.418,Z 279.917,A -85,B 0,C 180,E1 -10712.988,E2 -10712.988} C_VEL
LIN {X 0,Y 404.407,Z 279.924,A -85,B 0,C 180,E1 -10715.985,E2 -10715.985} C_VEL
LIN {X 0,Y 404.29,Z 279.933,A -85,B 0,C 180,E1 -10719.001,E2 -10719.001} C_VEL
LIN {X 0,Y 404.257,Z 279.941,A -85,B 0,C 180,E1 -10722.041,E2 -10722.041} C_VEL
LIN {X 0,Y 404.207,Z 279.944,A -85,B 0,C 180,E1 -10725.117,E2 -10725.117} C_VEL
LIN {X 0,Y 404.205,Z 279.947,A -85,B 0,C 180,E1 -10728.238,E2 -10728.238} C_VEL
LIN {X 0,Y 404.138,Z 279.952,A -85,B 0,C 180,E1 -10731.419,E2 -10731.419} C_VEL
LIN {X 0,Y 404.174,Z 279.953,A -85,B 0,C 180,E1 -10734.665,E2 -10734.665} C_VEL
LIN {X 0,Y 404.194,Z 279.945,A -85,B 0,C 180,E1 -10737.999,E2 -10737.999} C_VEL
LIN {X 0,Y 404.137,Z 279.954,A -85,B 0,C 180,E1 -10741.557,E2 -10741.557} C_VEL
LIN {X 0,Y 404.18,Z 279.952,A -85,B 0,C 180,E1 -10745.015,E2 -10745.015} C_VEL
LIN {X 0,Y 404.152,Z 279.952,A -85,B 0,C 180,E1 -10748.756,E2 -10748.756} C_VEL
LIN {X 0,Y 404.119,Z 279.959,A -85,B 0,C 180,E1 -10751.599,E2 -10751.599} C_VEL
LIN {X 0,Y 404.148,Z 279.95,A -85,B 0,C 180,E1 -10754.522,E2 -10754.522} C_VEL
LIN {X 0,Y 404.201,Z 279.948,A -85,B 0,C 180,E1 -10757.304,E2 -10757.304} C_VEL
LIN {X 0,Y 404.163,Z 279.953,A -85,B 0,C 180,E1 -10759.954,E2 -10759.954} C_VEL
LIN {X 0,Y 404.133,Z 279.953,A -85,B 0,C 180,E1 -10763.123,E2 -10763.123} C_VEL
LIN {X 0,Y 404.137,Z 279.956,A -85,B 0,C 180,E1 -10766.187,E2 -10766.187} C_VEL
LIN {X 0,Y 404.145,Z 279.954,A -85,B 0,C 180,E1 -10769.715,E2 -10769.715} C_VEL
LIN {X 0,Y 404.186,Z 279.945,A -85,B 0,C 180,E1 -10773.122,E2 -10773.122} C_VEL
LIN {X 0,Y 404.167,Z 279.948,A -85,B 0,C 180,E1 -10775.334,E2 -10775.334} C_VEL
LIN {X 0,Y 404.128,Z 279.958,A -85,B 0,C 180,E1 -10778.58,E2 -10778.58} C_VEL
LIN {X 0,Y 404.199,Z 279.945,A -85,B 0,C 180,E1 -10781.761,E2 -10781.761} C_VEL
LIN {X 0,Y 404.195,Z 279.948,A -85,B 0,C 180,E1 -10784.881,E2 -10784.881} C_VEL
LIN {X 0,Y 404.245,Z 279.939,A -85,B 0,C 180,E1 -10787.958,E2 -10787.958} C_VEL
LIN {X 0,Y 404.395,Z 279.92,A -85,B 0,C 180,E1 -10792.128,E2 -10792.128} C_VEL
LIN {X 0,Y 404.408,Z 279.918,A -85,B 0,C 180,E1 -10794.015,E2 -10794.015} C_VEL
LIN {X 0,Y 404.471,Z 279.91,A -85,B 0,C 180,E1 -10798.008,E2 -10798.008} C_VEL
LIN {X 0,Y 404.598,Z 279.894,A -85,B 0,C 180,E1 -10800,E2 -10800} C_VEL
LIN {X 0,Y 404.404,Z 279.923,A -85,B 0,C 180,E1 -10802.988,E2 -10802.988} C_VEL
LIN {X 0,Y 404.409,Z 279.919,A -85,B 0,C 180,E1 -10805.985,E2 -10805.985} C_VEL
LIN {X 0,Y 404.281,Z 279.936,A -85,B 0,C 180,E1 -10809.001,E2 -10809.001} C_VEL
LIN {X 0,Y 404.259,Z 279.938,A -85,B 0,C 180,E1 -10812.041,E2 -10812.041} C_VEL
LIN {X 0,Y 404.196,Z 279.946,A -85,B 0,C 180,E1 -10815.118,E2 -10815.118} C_VEL
LIN {X 0,Y 404.198,Z 279.946,A -85,B 0,C 180,E1 -10818.238,E2 -10818.238} C_VEL
LIN {X 0,Y 404.127,Z 279.955,A -85,B 0,C 180,E1 -10821.42,E2 -10821.42} C_VEL
LIN {X 0,Y 404.164,Z 279.949,A -85,B 0,C 180,E1 -10824.666,E2 -10824.666} C_VEL
LIN {X 0,Y 404.185,Z 279.952,A -85,B 0,C 180,E1 -10828,E2 -10828} C_VEL
LIN {X 0,Y 404.129,Z 279.953,A -85,B 0,C 180,E1 -10831.558,E2 -10831.558} C_VEL
LIN {X 0,Y 404.176,Z 279.948,A -85,B 0,C 180,E1 -10835.017,E2 -10835.017} C_VEL
LIN {X 0,Y 404.14,Z 279.955,A -85,B 0,C 180,E1 -10838.758,E2 -10838.758} C_VEL
LIN {X 0,Y 404.115,Z 279.954,A -85,B 0,C 180,E1 -10841.6,E2 -10841.6} C_VEL
LIN {X 0,Y 404.138,Z 279.957,A -85,B 0,C 180,E1 -10844.523,E2 -10844.523} C_VEL
LIN {X 0,Y 404.125,Z 279.955,A -85,B 0,C 180,E1 -10847.296,E2 -10847.296} C_VEL
LIN {X 0,Y 404.164,Z 279.948,A -85,B 0,C 180,E1 -10849.956,E2 -10849.956} C_VEL
LIN {X 0,Y 404.131,Z 279.958,A -85,B 0,C 180,E1 -10853.126,E2 -10853.126} C_VEL
LIN {X 0,Y 404.14,Z 279.951,A -85,B 0,C 180,E1 -10856.188,E2 -10856.188} C_VEL
LIN {X 0,Y 404.141,Z 279.953,A -85,B 0,C 180,E1 -10859.715,E2 -10859.715} C_VEL
LIN {X 0,Y 404.127,Z 279.96,A -85,B 0,C 180,E1 -10863.119,E2 -10863.119} C_VEL
LIN {X 0,Y 404.222,Z 280.048,A -85,B 0,C 180,E1 -10865.052,E2 -10865.052} C_VEL
LIN {X 0,Y 405.7,Z 288.267,A -85,B 0,C 180,E1 -10867.182,E2 -10867.182} C_VEL
LIN {X 0,Y 405.755,Z 293.212,A -85,B 0,C 180,E1 -10868.404,E2 -10868.404} C_VEL
LIN {X 0,Y 404.834,Z 308.48,A -85,B 0,C 180,E1 -10872.079,E2 -10872.079} C_VEL
LIN {X 0,Y 404.249,Z 319.247,A -85,B 0,C 180,E1 -10874.61,E2 -10874.61} C_VEL
LIN {X 0,Y 407.293,Z 342.646,A -85,B 0,C 180,E1 -10875.149,E2 -10875.149} C_VEL
LIN {X 0,Y 406.749,Z 395.947,A -85,B 0,C 180,E1 -10876.129,E2 -10876.129} C_VEL
LIN {X 0,Y 406.395,Z 405.74,A -85,B 0,C 180,E1 -10876.436,E2 -10876.436} C_VEL
LIN {X 0,Y 405.89,Z 417.42,A -85,B 0,C 180,E1 -10876.992,E2 -10876.992} C_VEL
LIN {X 0,Y 405.362,Z 428.133,A -85,B 0,C 180,E1 -10877.738,E2 -10877.738} C_VEL
LIN {X 0,Y 404.918,Z 436.503,A -85,B 0,C 180,E1 -10878.487,E2 -10878.487} C_VEL
LIN {X 0,Y 404.472,Z 444.421,A -85,B 0,C 180,E1 -10879.361,E2 -10879.361} C_VEL
LIN {X 0,Y 404.034,Z 450.962,A -85,B 0,C 180,E1 -10880.236,E2 -10880.236} C_VEL
LIN {X 0,Y 403.636,Z 457.185,A -85,B 0,C 180,E1 -10881.237,E2 -10881.237} C_VEL
LIN {X 0,Y 403.357,Z 462.35,A -85,B 0,C 180,E1 -10882.24,E2 -10882.24} C_VEL
LIN {X 0,Y 403.164,Z 466.896,A -85,B 0,C 180,E1 -10883.307,E2 -10883.307} C_VEL
LIN {X 0,Y 402.995,Z 470.978,A -85,B 0,C 180,E1 -10884.496,E2 -10884.496} C_VEL
LIN {X 0,Y 402.95,Z 473.717,A -85,B 0,C 180,E1 -10885.499,E2 -10885.499} C_VEL
LIN {X 0,Y 402.839,Z 476.701,A -85,B 0,C 180,E1 -10887,E2 -10887} C_VEL
LIN {X 0,Y 402.866,Z 478.023,A -85,B 0,C 180,E1 -10888.001,E2 -10888.001} C_VEL
LIN {X 0,Y 402.86,Z 478.862,A -85,B 0,C 180,E1 -10889,E2 -10889} C_VEL
LIN {X 0,Y 402.849,Z 479.171,A -85,B 0,C 180,E1 -10890,E2 -10890} C_VEL
LIN {X 0,Y 402.86,Z 478.901,A -85,B 0,C 180,E1 -10891,E2 -10891} C_VEL
LIN {X 0,Y 402.866,Z 478.161,A -85,B 0,C 180,E1 -10891.999,E2 -10891.999} C_VEL
LIN {X 0,Y 402.837,Z 476.943,A -85,B 0,C 180,E1 -10893,E2 -10893} C_VEL
LIN {X 0,Y 402.95,Z 474.063,A -85,B 0,C 180,E1 -10894.501,E2 -10894.501} C_VEL
LIN {X 0,Y 403.01,Z 471.449,A -85,B 0,C 180,E1 -10895.504,E2 -10895.504} C_VEL
LIN {X 0,Y 403.201,Z 467.45,A -85,B 0,C 180,E1 -10896.706,E2 -10896.706} C_VEL
LIN {X 0,Y 403.368,Z 463.112,A -85,B 0,C 180,E1 -10897.76,E2 -10897.76} C_VEL
LIN {X 0,Y 403.675,Z 458.134,A -85,B 0,C 180,E1 -10898.762,E2 -10898.762} C_VEL
LIN {X 0,Y 404.097,Z 452.139,A -85,B 0,C 180,E1 -10899.763,E2 -10899.763} C_VEL
LIN {X 0,Y 404.594,Z 444.846,A -85,B 0,C 180,E1 -10900.762,E2 -10900.762} C_VEL
LIN {X 0,Y 405.061,Z 437.058,A -85,B 0,C 180,E1 -10901.636,E2 -10901.636} C_VEL
LIN {X 0,Y 405.624,Z 428.866,A -85,B 0,C 180,E1 -10902.381,E2 -10902.381} C_VEL
LIN {X 0,Y 406.069,Z 420.346,A -85,B 0,C 180,E1 -10903.002,E2 -10903.002} C_VEL
LIN {X 0,Y 406.498,Z 410.398,A -85,B 0,C 180,E1 -10903.561,E2 -10903.561} C_VEL
LIN {X 0,Y 407.046,Z 397.794,A -85,B 0,C 180,E1 -10904.022,E2 -10904.022} C_VEL
LIN {X 0,Y 407.401,Z 374.135,A -85,B 0,C 180,E1 -10904.484,E2 -10904.484} C_VEL
LIN {X 0,Y 407.6,Z 341.49,A -85,B 0,C 180,E1 -10905.078,E2 -10905.078} C_VEL
LIN {X 0,Y 404.319,Z 318.491,A -85,B 0,C 180,E1 -10905.652,E2 -10905.652} C_VEL
LIN {X 0,Y 405.166,Z 303.07,A -85,B 0,C 180,E1 -10909.242,E2 -10909.242} C_VEL
LIN {X 0,Y 405.9,Z 289.747,A -85,B 0,C 180,E1 -10912.39,E2 -10912.39} C_VEL
LIN {X 0,Y 404.207,Z 279.95,A -85,B 0,C 180,E1 -10914.901,E2 -10914.901} C_VEL
LIN {X 0,Y 404.114,Z 279.96,A -85,B 0,C 180,E1 -10918.005,E2 -10918.005} C_VEL
LIN {X 0,Y 404.14,Z 279.959,A -85,B 0,C 180,E1 -10920.285,E2 -10920.285} C_VEL
LIN {X 0,Y 404.14,Z 279.954,A -85,B 0,C 180,E1 -10923.812,E2 -10923.812} C_VEL
LIN {X 0,Y 404.13,Z 279.96,A -85,B 0,C 180,E1 -10926.874,E2 -10926.874} C_VEL
LIN {X 0,Y 404.142,Z 279.957,A -85,B 0,C 180,E1 -10930.079,E2 -10930.079} C_VEL
LIN {X 0,Y 404.143,Z 279.959,A -85,B 0,C 180,E1 -10933.082,E2 -10933.082} C_VEL
LIN {X 0,Y 404.14,Z 279.956,A -85,B 0,C 180,E1 -10935.925,E2 -10935.925} C_VEL
LIN {X 0,Y 404.11,Z 279.955,A -85,B 0,C 180,E1 -10938.634,E2 -10938.634} C_VEL
LIN {X 0,Y 404.14,Z 279.957,A -85,B 0,C 180,E1 -10941.492,E2 -10941.492} C_VEL
LIN {X 0,Y 404.176,Z 279.949,A -85,B 0,C 180,E1 -10944.983,E2 -10944.983} C_VEL
LIN {X 0,Y 404.132,Z 279.952,A -85,B 0,C 180,E1 -10948.553,E2 -10948.553} C_VEL
LIN {X 0,Y 404.185,Z 279.944,A -85,B 0,C 180,E1 -10952,E2 -10952} C_VEL
LIN {X 0,Y 404.163,Z 279.95,A -85,B 0,C 180,E1 -10955.334,E2 -10955.334} C_VEL
LIN {X 0,Y 404.126,Z 279.951,A -85,B 0,C 180,E1 -10958.58,E2 -10958.58} C_VEL
LIN {X 0,Y 404.198,Z 279.947,A -85,B 0,C 180,E1 -10961.761,E2 -10961.761} C_VEL
LIN {X 0,Y 404.193,Z 279.943,A -85,B 0,C 180,E1 -10964.882,E2 -10964.882} C_VEL
LIN {X 0,Y 404.245,Z 279.941,A -85,B 0,C 180,E1 -10967.958,E2 -10967.958} C_VEL
LIN {X 0,Y 404.394,Z 279.916,A -85,B 0,C 180,E1 -10972.128,E2 -10972.128} C_VEL
LIN {X 0,Y 404.409,Z 279.918,A -85,B 0,C 180,E1 -10974.015,E2 -10974.015} C_VEL
LIN {X 0,Y 404.467,Z 279.907,A -85,B 0,C 180,E1 -10978.009,E2 -10978.009} C_VEL
LIN {X 0,Y 404.598,Z 279.894,A -85,B 0,C 180,E1 -10980,E2 -10980} C_VEL
LIN {X 0,Y 404.404,Z 279.916,A -85,B 0,C 180,E1 -10982.989,E2 -10982.989} C_VEL
LIN {X 0,Y 404.357,Z 279.926,A -85,B 0,C 180,E1 -10986.988,E2 -10986.988} C_VEL
LIN {X 0,Y 404.246,Z 279.94,A -85,B 0,C 180,E1 -10990.012,E2 -10990.012} C_VEL
LIN {X 0,Y 404.255,Z 279.937,A -85,B 0,C 180,E1 -10993.212,E2 -10993.212} C_VEL
LIN {X 0,Y 404.205,Z 279.943,A -85,B 0,C 180,E1 -10997.008,E2 -10997.008} C_VEL
LIN {X 0,Y 404.153,Z 279.951,A -85,B 0,C 180,E1 -11000.352,E2 -11000.352} C_VEL
LIN {X 0,Y 404.159,Z 279.956,A -85,B 0,C 180,E1 -11003.575,E2 -11003.575} C_VEL
LIN {X 0,Y 404.174,Z 279.956,A -85,B 0,C 180,E1 -11005.767,E2 -11005.767} C_VEL
LIN {X 0,Y 404.189,Z 279.952,A -85,B 0,C 180,E1 -11008,E2 -11008} C_VEL
LIN {X 0,Y 404.134,Z 279.955,A -85,B 0,C 180,E1 -11011.56,E2 -11011.56} C_VEL
LIN {X 0,Y 404.178,Z 279.946,A -85,B 0,C 180,E1 -11015.017,E2 -11015.017} C_VEL
LIN {X 0,Y 404.156,Z 279.955,A -85,B 0,C 180,E1 -11018.757,E2 -11018.757} C_VEL
LIN {X 0,Y 404.237,Z 280.084,A -85,B 0,C 180,E1 -11022.031,E2 -11022.031} C_VEL
LIN {X 0,Y 405.014,Z 284.629,A -85,B 0,C 180,E1 -11023.216,E2 -11023.216} C_VEL
LIN {X 0,Y 404.706,Z 295.905,A -85,B 0,C 180,E1 -11026.004,E2 -11026.004} C_VEL
LIN {X 0,Y 404.667,Z 297.75,A -85,B 0,C 180,E1 -11026.425,E2 -11026.425} C_VEL
LIN {X 0,Y 407.851,Z 314.752,A -85,B 0,C 180,E1 -11026.877,E2 -11026.877} C_VEL
LIN {X 0,Y 407.162,Z 374.361,A -85,B 0,C 180,E1 -11027.979,E2 -11027.979} C_VEL
LIN {X 0,Y 406.913,Z 384.377,A -85,B 0,C 180,E1 -11028.302,E2 -11028.302} C_VEL
LIN {X 0,Y 406.566,Z 395.717,A -85,B 0,C 180,E1 -11028.857,E2 -11028.857} C_VEL
LIN {X 0,Y 405.991,Z 406.435,A -85,B 0,C 180,E1 -11029.612,E2 -11029.612} C_VEL
LIN {X 0,Y 405.588,Z 413.984,A -85,B 0,C 180,E1 -11030.287,E2 -11030.287} C_VEL
LIN {X 0,Y 405.136,Z 420.945,A -85,B 0,C 180,E1 -11031.037,E2 -11031.037} C_VEL
LIN {X 0,Y 404.622,Z 427.837,A -85,B 0,C 180,E1 -11031.932,E2 -11031.932} C_VEL
LIN {X 0,Y 404.28,Z 433.836,A -85,B 0,C 180,E1 -11032.873,E2 -11032.873} C_VEL
LIN {X 0,Y 403.845,Z 439.917,A -85,B 0,C 180,E1 -11034.033,E2 -11034.033} C_VEL
LIN {X 0,Y 403.5,Z 444.961,A -85,B 0,C 180,E1 -11035.225,E2 -11035.225} C_VEL
LIN {X 0,Y 403.17,Z 450.116,A -85,B 0,C 180,E1 -11036.797,E2 -11036.797} C_VEL
LIN {X 0,Y 402.961,Z 453.794,A -85,B 0,C 180,E1 -11038.452,E2 -11038.452} C_VEL
LIN {X 0,Y 402.834,Z 455.516,A -85,B 0,C 180,E1 -11039.607,E2 -11039.607} C_VEL
LIN {X 0,Y 402.714,Z 456.555,A -85,B 0,C 180,E1 -11040.76,E2 -11040.76} C_VEL
LIN {X 0,Y 402.665,Z 456.902,A -85,B 0,C 180,E1 -11041.886,E2 -11041.886} C_VEL
LIN {X 0,Y 402.706,Z 456.58,A -85,B 0,C 180,E1 -11043.016,E2 -11043.016} C_VEL
LIN {X 0,Y 402.73,Z 455.636,A -85,B 0,C 180,E1 -11044.135,E2 -11044.135} C_VEL
LIN {X 0,Y 402.953,Z 453.118,A -85,B 0,C 180,E1 -11045.804,E2 -11045.804} C_VEL
LIN {X 0,Y 403.109,Z 450.579,A -85,B 0,C 180,E1 -11046.905,E2 -11046.905} C_VEL
LIN {X 0,Y 403.294,Z 447.247,A -85,B 0,C 180,E1 -11048.02,E2 -11048.02} C_VEL
LIN {X 0,Y 403.626,Z 440.939,A -85,B 0,C 180,E1 -11049.621,E2 -11049.621} C_VEL
LIN {X 0,Y 403.963,Z 435.536,A -85,B 0,C 180,E1 -11050.698,E2 -11050.698} C_VEL
LIN {X 0,Y 404.398,Z 428.949,A -85,B 0,C 180,E1 -11051.771,E2 -11051.771} C_VEL
LIN {X 0,Y 404.815,Z 421.873,A -85,B 0,C 180,E1 -11052.719,E2 -11052.719} C_VEL
LIN {X 0,Y 405.251,Z 414.782,A -85,B 0,C 180,E1 -11053.503,E2 -11053.503} C_VEL
LIN {X 0,Y 405.666,Z 407.537,A -85,B 0,C 180,E1 -11054.166,E2 -11054.166} C_VEL
LIN {X 0,Y 406.086,Z 398.599,A -85,B 0,C 180,E1 -11054.826,E2 -11054.826} C_VEL
LIN {X 0,Y 406.405,Z 388.574,A -85,B 0,C 180,E1 -11055.393,E2 -11055.393} C_VEL
LIN {X 0,Y 406.8,Z 376.397,A -85,B 0,C 180,E1 -11055.848,E2 -11055.848} C_VEL
LIN {X 0,Y 407.064,Z 355.873,A -85,B 0,C 180,E1 -11056.256,E2 -11056.256} C_VEL
LIN {X 0,Y 407.35,Z 314.786,A -85,B 0,C 180,E1 -11056.997,E2 -11056.997} C_VEL
LIN {X 0,Y 404.482,Z 297.873,A -85,B 0,C 180,E1 -11057.424,E2 -11057.424} C_VEL
LIN {X 0,Y 404.918,Z 286.564,A -85,B 0,C 180,E1 -11060.51,E2 -11060.51} C_VEL
LIN {X 0,Y 404.788,Z 282.599,A -85,B 0,C 180,E1 -11061.616,E2 -11061.616} C_VEL
LIN {X 0,Y 404.328,Z 281.255,A -85,B 0,C 180,E1 -11062.125,E2 -11062.125} C_VEL
LIN {X 0,Y 403.372,Z 280.569,A -85,B 0,C 180,E1 -11062.652,E2 -11062.652} C_VEL
LIN {X 0,Y 400.75,Z 280.381,A -85,B 0,C 180,E1 -11063.719,E2 -11063.719} C_VEL
LIN {X 0,Y 398.211,Z 280.691,A -85,B 0,C 180,E1 -11064.83,E2 -11064.83} C_VEL
LIN {X 0,Y 397.205,Z 280.823,A -85,B 0,C 180,E1 -11065.692,E2 -11065.692} C_VEL
LIN {X 0,Y 397.162,Z 280.826,A -85,B 0,C 180,E1 -11065.984,E2 -11065.984} C_VEL
LIN {X 0,Y 397.451,Z 280.791,A -85,B 0,C 180,E1 -11067.973,E2 -11067.973} C_VEL
LIN {X 0,Y 397.581,Z 280.775,A -85,B 0,C 180,E1 -11070,E2 -11070} C_VEL
LIN {X 0,Y 397.377,Z 280.794,A -85,B 0,C 180,E1 -11073.041,E2 -11073.041} C_VEL
LIN {X 0,Y 397.357,Z 280.804,A -85,B 0,C 180,E1 -11076.092,E2 -11076.092} C_VEL
LIN {X 0,Y 397.253,Z 280.809,A -85,B 0,C 180,E1 -11079.162,E2 -11079.162} C_VEL
LIN {X 0,Y 397.22,Z 280.82,A -85,B 0,C 180,E1 -11082.258,E2 -11082.258} C_VEL
LIN {X 0,Y 397.18,Z 280.818,A -85,B 0,C 180,E1 -11085.392,E2 -11085.392} C_VEL
LIN {X 0,Y 397.158,Z 280.829,A -85,B 0,C 180,E1 -11088.573,E2 -11088.573} C_VEL
LIN {X 0,Y 397.096,Z 280.829,A -85,B 0,C 180,E1 -11091.818,E2 -11091.818} C_VEL
LIN {X 0,Y 397.152,Z 280.823,A -85,B 0,C 180,E1 -11095.511,E2 -11095.511} C_VEL
LIN {X 0,Y 397.121,Z 280.829,A -85,B 0,C 180,E1 -11098.543,E2 -11098.543} C_VEL
LIN {X 0,Y 397.075,Z 280.831,A -85,B 0,C 180,E1 -11102.071,E2 -11102.071} C_VEL
LIN {X 0,Y 397.115,Z 280.83,A -85,B 0,C 180,E1 -11105.502,E2 -11105.502} C_VEL
LIN {X 0,Y 397.127,Z 280.828,A -85,B 0,C 180,E1 -11108.861,E2 -11108.861} C_VEL
LIN {X 0,Y 397.064,Z 280.833,A -85,B 0,C 180,E1 -11112.266,E2 -11112.266} C_VEL
LIN {X 0,Y 397.11,Z 280.829,A -85,B 0,C 180,E1 -11115.064,E2 -11115.064} C_VEL
LIN {X 0,Y 397.15,Z 280.825,A -85,B 0,C 180,E1 -11118.006,E2 -11118.006} C_VEL
LIN {X 0,Y 397.102,Z 280.836,A -85,B 0,C 180,E1 -11121.725,E2 -11121.725} C_VEL
LIN {X 0,Y 397.118,Z 280.829,A -85,B 0,C 180,E1 -11125.506,E2 -11125.506} C_VEL
LIN {X 0,Y 397.075,Z 280.831,A -85,B 0,C 180,E1 -11129.117,E2 -11129.117} C_VEL
LIN {X 0,Y 397.186,Z 280.82,A -85,B 0,C 180,E1 -11132.609,E2 -11132.609} C_VEL
LIN {X 0,Y 397.123,Z 280.83,A -85,B 0,C 180,E1 -11135.981,E2 -11135.981} C_VEL
LIN {X 0,Y 397.129,Z 280.826,A -85,B 0,C 180,E1 -11139.704,E2 -11139.704} C_VEL
LIN {X 0,Y 397.172,Z 280.823,A -85,B 0,C 180,E1 -11142.844,E2 -11142.844} C_VEL
LIN {X 0,Y 397.218,Z 280.821,A -85,B 0,C 180,E1 -11146.702,E2 -11146.702} C_VEL
LIN {X 0,Y 397.206,Z 280.815,A -85,B 0,C 180,E1 -11149.809,E2 -11149.809} C_VEL
LIN {X 0,Y 397.343,Z 280.806,A -85,B 0,C 180,E1 -11152.888,E2 -11152.888} C_VEL
LIN {X 0,Y 397.241,Z 280.819,A -85,B 0,C 180,E1 -11154.925,E2 -11154.925} C_VEL
LIN {X 0,Y 397.439,Z 280.786,A -85,B 0,C 180,E1 -11157.973,E2 -11157.973} C_VEL
LIN {X 0,Y 397.568,Z 280.77,A -85,B 0,C 180,E1 -11160,E2 -11160} C_VEL
LIN {X 0,Y 397.364,Z 280.801,A -85,B 0,C 180,E1 -11163.041,E2 -11163.041} C_VEL
LIN {X 0,Y 397.36,Z 280.796,A -85,B 0,C 180,E1 -11166.092,E2 -11166.092} C_VEL
LIN {X 0,Y 397.243,Z 280.815,A -85,B 0,C 180,E1 -11169.162,E2 -11169.162} C_VEL
LIN {X 0,Y 397.218,Z 280.814,A -85,B 0,C 180,E1 -11172.258,E2 -11172.258} C_VEL
LIN {X 0,Y 397.168,Z 280.824,A -85,B 0,C 180,E1 -11175.392,E2 -11175.392} C_VEL
LIN {X 0,Y 397.151,Z 280.822,A -85,B 0,C 180,E1 -11178.574,E2 -11178.574} C_VEL
LIN {X 0,Y 397.085,Z 280.837,A -85,B 0,C 180,E1 -11181.819,E2 -11181.819} C_VEL
LIN {X 0,Y 397.143,Z 280.825,A -85,B 0,C 180,E1 -11185.513,E2 -11185.513} C_VEL
LIN {X 0,Y 397.112,Z 280.829,A -85,B 0,C 180,E1 -11188.544,E2 -11188.544} C_VEL
LIN {X 0,Y 397.069,Z 280.838,A -85,B 0,C 180,E1 -11192.072,E2 -11192.072} C_VEL
LIN {X 0,Y 397.111,Z 280.827,A -85,B 0,C 180,E1 -11195.504,E2 -11195.504} C_VEL
LIN {X 0,Y 397.117,Z 280.829,A -85,B 0,C 180,E1 -11198.861,E2 -11198.861} C_VEL
LIN {X 0,Y 397.061,Z 280.837,A -85,B 0,C 180,E1 -11202.268,E2 -11202.268} C_VEL
LIN {X 0,Y 397.08,Z 280.834,A -85,B 0,C 180,E1 -11205.07,E2 -11205.07} C_VEL
LIN {X 0,Y 397.055,Z 280.834,A -85,B 0,C 180,E1 -11208.023,E2 -11208.023} C_VEL
LIN {X 0,Y 397.121,Z 280.831,A -85,B 0,C 180,E1 -11211.14,E2 -11211.14} C_VEL
LIN {X 0,Y 397.114,Z 280.828,A -85,B 0,C 180,E1 -11214.498,E2 -11214.498} C_VEL
LIN {X 0,Y 397.074,Z 280.832,A -85,B 0,C 180,E1 -11217.929,E2 -11217.929} C_VEL
LIN {X 0,Y 397.114,Z 280.826,A -85,B 0,C 180,E1 -11220.296,E2 -11220.296} C_VEL
LIN {X 0,Y 397.089,Z 280.835,A -85,B 0,C 180,E1 -11223.739,E2 -11223.739} C_VEL
LIN {X 0,Y 397.159,Z 280.912,A -85,B 0,C 180,E1 -11224.869,E2 -11224.869} C_VEL
LIN {X 0,Y 398.731,Z 289.684,A -85,B 0,C 180,E1 -11227.185,E2 -11227.185} C_VEL
LIN {X 0,Y 398.738,Z 295.094,A -85,B 0,C 180,E1 -11228.541,E2 -11228.541} C_VEL
LIN {X 0,Y 397.695,Z 311.356,A -85,B 0,C 180,E1 -11232.518,E2 -11232.518} C_VEL
LIN {X 0,Y 397.256,Z 318.917,A -85,B 0,C 180,E1 -11234.349,E2 -11234.349} C_VEL
LIN {X 0,Y 400.391,Z 342.983,A -85,B 0,C 180,E1 -11234.914,E2 -11234.914} C_VEL
LIN {X 0,Y 399.83,Z 396.33,A -85,B 0,C 180,E1 -11235.917,E2 -11235.917} C_VEL
LIN {X 0,Y 399.43,Z 406.743,A -85,B 0,C 180,E1 -11236.259,E2 -11236.259} C_VEL
LIN {X 0,Y 398.893,Z 418.91,A -85,B 0,C 180,E1 -11236.889,E2 -11236.889} C_VEL
LIN {X 0,Y 398.433,Z 427.732,A -85,B 0,C 180,E1 -11237.522,E2 -11237.522} C_VEL
LIN {X 0,Y 397.941,Z 436.139,A -85,B 0,C 180,E1 -11238.282,E2 -11238.282} C_VEL
LIN {X 0,Y 397.501,Z 444.087,A -85,B 0,C 180,E1 -11239.173,E2 -11239.173} C_VEL
LIN {X 0,Y 397.019,Z 450.651,A -85,B 0,C 180,E1 -11240.062,E2 -11240.062} C_VEL
LIN {X 0,Y 396.606,Z 456.894,A -85,B 0,C 180,E1 -11241.08,E2 -11241.08} C_VEL
LIN {X 0,Y 396.295,Z 462.076,A -85,B 0,C 180,E1 -11242.1,E2 -11242.1} C_VEL
LIN {X 0,Y 396.123,Z 466.487,A -85,B 0,C 180,E1 -11243.148,E2 -11243.148} C_VEL
LIN {X 0,Y 395.899,Z 470.732,A -85,B 0,C 180,E1 -11244.397,E2 -11244.397} C_VEL
LIN {X 0,Y 395.881,Z 473.485,A -85,B 0,C 180,E1 -11245.418,E2 -11245.418} C_VEL
LIN {X 0,Y 395.742,Z 476.479,A -85,B 0,C 180,E1 -11246.946,E2 -11246.946} C_VEL
LIN {X 0,Y 395.765,Z 477.811,A -85,B 0,C 180,E1 -11247.965,E2 -11247.965} C_VEL
LIN {X 0,Y 395.789,Z 478.662,A -85,B 0,C 180,E1 -11248.983,E2 -11248.983} C_VEL
LIN {X 0,Y 395.776,Z 478.971,A -85,B 0,C 180,E1 -11250,E2 -11250} C_VEL
LIN {X 0,Y 395.789,Z 478.709,A -85,B 0,C 180,E1 -11251.017,E2 -11251.017} C_VEL
LIN {X 0,Y 395.764,Z 477.977,A -85,B 0,C 180,E1 -11252.035,E2 -11252.035} C_VEL
LIN {X 0,Y 395.741,Z 476.768,A -85,B 0,C 180,E1 -11253.054,E2 -11253.054} C_VEL
LIN {X 0,Y 395.881,Z 473.896,A -85,B 0,C 180,E1 -11254.582,E2 -11254.582} C_VEL
LIN {X 0,Y 395.948,Z 469.753,A -85,B 0,C 180,E1 -11256.113,E2 -11256.113} C_VEL
LIN {X 0,Y 396.248,Z 464.149,A -85,B 0,C 180,E1 -11257.644,E2 -11257.644} C_VEL
LIN {X 0,Y 396.638,Z 458.016,A -85,B 0,C 180,E1 -11258.919,E2 -11258.919} C_VEL
LIN {X 0,Y 397.077,Z 452.042,A -85,B 0,C 180,E1 -11259.937,E2 -11259.937} C_VEL
LIN {X 0,Y 397.63,Z 444.777,A -85,B 0,C 180,E1 -11260.953,E2 -11260.953} C_VEL
LIN {X 0,Y 398.092,Z 437.023,A -85,B 0,C 180,E1 -11261.843,E2 -11261.843} C_VEL
LIN {X 0,Y 398.683,Z 428.873,A -85,B 0,C 180,E1 -11262.6,E2 -11262.6} C_VEL
LIN {X 0,Y 399.169,Z 420.413,A -85,B 0,C 180,E1 -11263.231,E2 -11263.231} C_VEL
LIN {X 0,Y 399.624,Z 410.543,A -85,B 0,C 180,E1 -11263.799,E2 -11263.799} C_VEL
LIN {X 0,Y 400.179,Z 398.35,A -85,B 0,C 180,E1 -11264.267,E2 -11264.267} C_VEL
LIN {X 0,Y 400.51,Z 378.782,A -85,B 0,C 180,E1 -11264.667,E2 -11264.667} C_VEL
LIN {X 0,Y 400.703,Z 341.536,A -85,B 0,C 180,E1 -11265.36,E2 -11265.36} C_VEL
LIN {X 0,Y 397.358,Z 318.221,A -85,B 0,C 180,E1 -11265.967,E2 -11265.967} C_VEL
LIN {X 0,Y 398.163,Z 304.06,A -85,B 0,C 180,E1 -11269.326,E2 -11269.326} C_VEL
LIN {X 0,Y 398.912,Z 291.851,A -85,B 0,C 180,E1 -11272.258,E2 -11272.258} C_VEL
LIN {X 0,Y 397.973,Z 285.149,A -85,B 0,C 180,E1 -11273.964,E2 -11273.964} C_VEL
LIN {X 0,Y 397.138,Z 280.831,A -85,B 0,C 180,E1 -11275.132,E2 -11275.132} C_VEL
LIN {X 0,Y 397.067,Z 280.84,A -85,B 0,C 180,E1 -11278.547,E2 -11278.547} C_VEL
LIN {X 0,Y 397.077,Z 280.833,A -85,B 0,C 180,E1 -11281.835,E2 -11281.835} C_VEL
LIN {X 0,Y 397.12,Z 280.831,A -85,B 0,C 180,E1 -11284.493,E2 -11284.493} C_VEL
LIN {X 0,Y 397.094,Z 280.835,A -85,B 0,C 180,E1 -11288.275,E2 -11288.275} C_VEL
LIN {X 0,Y 397.08,Z 280.841,A -85,B 0,C 180,E1 -11290.908,E2 -11290.908} C_VEL
LIN {X 0,Y 397.093,Z 280.837,A -85,B 0,C 180,E1 -11293.648,E2 -11293.648} C_VEL
LIN {X 0,Y 397.095,Z 280.832,A -85,B 0,C 180,E1 -11296.52,E2 -11296.52} C_VEL
LIN {X 0,Y 397.104,Z 280.83,A -85,B 0,C 180,E1 -11300.422,E2 -11300.422} C_VEL
LIN {X 0,Y 397.099,Z 280.831,A -85,B 0,C 180,E1 -11304.265,E2 -11304.265} C_VEL
LIN {X 0,Y 397.105,Z 280.825,A -85,B 0,C 180,E1 -11306.726,E2 -11306.726} C_VEL
LIN {X 0,Y 397.114,Z 280.829,A -85,B 0,C 180,E1 -11310.295,E2 -11310.295} C_VEL
LIN {X 0,Y 397.184,Z 280.812,A -85,B 0,C 180,E1 -11312.609,E2 -11312.609} C_VEL
LIN {X 0,Y 397.117,Z 280.833,A -85,B 0,C 180,E1 -11315.981,E2 -11315.981} C_VEL
LIN {X 0,Y 397.128,Z 280.822,A -85,B 0,C 180,E1 -11319.704,E2 -11319.704} C_VEL
LIN {X 0,Y 397.171,Z 280.818,A -85,B 0,C 180,E1 -11322.845,E2 -11322.845} C_VEL
LIN {X 0,Y 397.217,Z 280.819,A -85,B 0,C 180,E1 -11326.702,E2 -11326.702} C_VEL
LIN {X 0,Y 397.206,Z 280.812,A -85,B 0,C 180,E1 -11329.809,E2 -11329.809} C_VEL
LIN {X 0,Y 397.343,Z 280.803,A -85,B 0,C 180,E1 -11332.888,E2 -11332.888} C_VEL
LIN {X 0,Y 397.241,Z 280.811,A -85,B 0,C 180,E1 -11334.925,E2 -11334.925} C_VEL
LIN {X 0,Y 397.436,Z 280.782,A -85,B 0,C 180,E1 -11337.973,E2 -11337.973} C_VEL
LIN {X 0,Y 397.567,Z 280.77,A -85,B 0,C 180,E1 -11340,E2 -11340} C_VEL
LIN {X 0,Y 397.363,Z 280.793,A -85,B 0,C 180,E1 -11343.042,E2 -11343.042} C_VEL
LIN {X 0,Y 397.306,Z 280.8,A -85,B 0,C 180,E1 -11346.501,E2 -11346.501} C_VEL
LIN {X 0,Y 397.24,Z 280.813,A -85,B 0,C 180,E1 -11349.162,E2 -11349.162} C_VEL
LIN {X 0,Y 397.207,Z 280.81,A -85,B 0,C 180,E1 -11352.259,E2 -11352.259} C_VEL
LIN {X 0,Y 397.167,Z 280.827,A -85,B 0,C 180,E1 -11355.393,E2 -11355.393} C_VEL
LIN {X 0,Y 397.151,Z 280.826,A -85,B 0,C 180,E1 -11358.574,E2 -11358.574} C_VEL
LIN {X 0,Y 397.086,Z 280.84,A -85,B 0,C 180,E1 -11361.819,E2 -11361.819} C_VEL
LIN {X 0,Y 397.147,Z 280.826,A -85,B 0,C 180,E1 -11365.132,E2 -11365.132} C_VEL
LIN {X 0,Y 397.155,Z 280.828,A -85,B 0,C 180,E1 -11367.777,E2 -11367.777} C_VEL
LIN {X 0,Y 397.075,Z 280.833,A -85,B 0,C 180,E1 -11370.883,E2 -11370.883} C_VEL
LIN {X 0,Y 397.118,Z 280.828,A -85,B 0,C 180,E1 -11374.494,E2 -11374.494} C_VEL
LIN {X 0,Y 397.102,Z 280.836,A -85,B 0,C 180,E1 -11378.275,E2 -11378.275} C_VEL
LIN {X 0,Y 397.179,Z 281.015,A -85,B 0,C 180,E1 -11381.833,E2 -11381.833} C_VEL
LIN {X 0,Y 398.081,Z 286.029,A -85,B 0,C 180,E1 -11383.167,E2 -11383.167} C_VEL
LIN {X 0,Y 397.686,Z 297.699,A -85,B 0,C 180,E1 -11386.099,E2 -11386.099} C_VEL
LIN {X 0,Y 401.042,Z 315.532,A -85,B 0,C 180,E1 -11386.604,E2 -11386.604} C_VEL
LIN {X 0,Y 400.343,Z 374.418,A -85,B 0,C 180,E1 -11387.712,E2 -11387.712} C_VEL
LIN {X 0,Y 400.041,Z 384.112,A -85,B 0,C 180,E1 -11388.025,E2 -11388.025} C_VEL
LIN {X 0,Y 399.741,Z 395.112,A -85,B 0,C 180,E1 -11388.562,E2 -11388.562} C_VEL
LIN {X 0,Y 399.13,Z 406.286,A -85,B 0,C 180,E1 -11389.346,E2 -11389.346} C_VEL
LIN {X 0,Y 398.622,Z 414.675,A -85,B 0,C 180,E1 -11390.111,E2 -11390.111} C_VEL
LIN {X 0,Y 398.134,Z 422.229,A -85,B 0,C 180,E1 -11390.96,E2 -11390.96} C_VEL
LIN {X 0,Y 397.632,Z 428.379,A -85,B 0,C 180,E1 -11391.787,E2 -11391.787} C_VEL
LIN {X 0,Y 397.261,Z 434.408,A -85,B 0,C 180,E1 -11392.76,E2 -11392.76} C_VEL
LIN {X 0,Y 396.813,Z 440.343,A -85,B 0,C 180,E1 -11393.923,E2 -11393.923} C_VEL
LIN {X 0,Y 396.493,Z 444.903,A -85,B 0,C 180,E1 -11395.019,E2 -11395.019} C_VEL
LIN {X 0,Y 396.106,Z 450.153,A -85,B 0,C 180,E1 -11396.633,E2 -11396.633} C_VEL
LIN {X 0,Y 396.006,Z 452.979,A -85,B 0,C 180,E1 -11397.832,E2 -11397.832} C_VEL
LIN {X 0,Y 395.822,Z 454.996,A -85,B 0,C 180,E1 -11399.01,E2 -11399.01} C_VEL
LIN {X 0,Y 395.63,Z 456.613,A -85,B 0,C 180,E1 -11400.51,E2 -11400.51} C_VEL
LIN {X 0,Y 395.586,Z 456.949,A -85,B 0,C 180,E1 -11402.49,E2 -11402.49} C_VEL
LIN {X 0,Y 395.606,Z 456.333,A -85,B 0,C 180,E1 -11403.633,E2 -11403.633} C_VEL
LIN {X 0,Y 395.74,Z 454.855,A -85,B 0,C 180,E1 -11404.92,E2 -11404.92} C_VEL
LIN {X 0,Y 395.871,Z 453.219,A -85,B 0,C 180,E1 -11405.901,E2 -11405.901} C_VEL
LIN {X 0,Y 396.073,Z 449.794,A -85,B 0,C 180,E1 -11407.324,E2 -11407.324} C_VEL
LIN {X 0,Y 396.339,Z 445.39,A -85,B 0,C 180,E1 -11408.685,E2 -11408.685} C_VEL
LIN {X 0,Y 396.625,Z 440.357,A -85,B 0,C 180,E1 -11409.907,E2 -11409.907} C_VEL
LIN {X 0,Y 397.047,Z 433.949,A -85,B 0,C 180,E1 -11411.154,E2 -11411.154} C_VEL
LIN {X 0,Y 397.518,Z 427.016,A -85,B 0,C 180,E1 -11412.244,E2 -11412.244} C_VEL
LIN {X 0,Y 398.16,Z 417.146,A -85,B 0,C 180,E1 -11413.464,E2 -11413.464} C_VEL
LIN {X 0,Y 398.648,Z 408.786,A -85,B 0,C 180,E1 -11414.273,E2 -11414.273} C_VEL
LIN {X 0,Y 399.053,Z 400.774,A -85,B 0,C 180,E1 -11414.9,E2 -11414.9} C_VEL
LIN {X 0,Y 399.414,Z 391.515,A -85,B 0,C 180,E1 -11415.465,E2 -11415.465} C_VEL
LIN {X 0,Y 399.687,Z 382.328,A -85,B 0,C 180,E1 -11415.879,E2 -11415.879} C_VEL
LIN {X 0,Y 399.951,Z 372.238,A -85,B 0,C 180,E1 -11416.181,E2 -11416.181} C_VEL
LIN {X 0,Y 400.4,Z 314.953,A -85,B 0,C 180,E1 -11417.246,E2 -11417.246} C_VEL
LIN {X 0,Y 397.459,Z 298.068,A -85,B 0,C 180,E1 -11417.685,E2 -11417.685} C_VEL
LIN {X 0,Y 397.912,Z 286.62,A -85,B 0,C 180,E1 -11420.854,E2 -11420.854} C_VEL
LIN {X 0,Y 397.449,Z 281.316,A -85,B 0,C 180,E1 -11422.38,E2 -11422.38} C_VEL
LIN {X 0,Y 397.351,Z 280.803,A -85,B 0,C 180,E1 -11422.633,E2 -11422.633} C_VEL
LIN {X 0,Y 397.254,Z 280.81,A -85,B 0,C 180,E1 -11424.925,E2 -11424.925} C_VEL
LIN {X 0,Y 397.162,Z 280.826,A -85,B 0,C 180,E1 -11425.984,E2 -11425.984} C_VEL
LIN {X 0,Y 396.648,Z 280.885,A -85,B 0,C 180,E1 -11426.831,E2 -11426.831} C_VEL
LIN {X 0,Y 394.016,Z 281.216,A -85,B 0,C 180,E1 -11428.213,E2 -11428.213} C_VEL
LIN {X 0,Y 390.834,Z 281.617,A -85,B 0,C 180,E1 -11429.899,E2 -11429.899} C_VEL
LIN {X 0,Y 390.441,Z 281.659,A -85,B 0,C 180,E1 -11430.479,E2 -11430.479} C_VEL
LIN {X 0,Y 390.312,Z 281.674,A -85,B 0,C 180,E1 -11433.096,E2 -11433.096} C_VEL
LIN {X 0,Y 390.31,Z 281.681,A -85,B 0,C 180,E1 -11436.202,E2 -11436.202} C_VEL
LIN {X 0,Y 390.205,Z 281.687,A -85,B 0,C 180,E1 -11439.328,E2 -11439.328} C_VEL
LIN {X 0,Y 390.196,Z 281.688,A -85,B 0,C 180,E1 -11443.438,E2 -11443.438} C_VEL
LIN {X 0,Y 390.129,Z 281.697,A -85,B 0,C 180,E1 -11447.298,E2 -11447.298} C_VEL
LIN {X 0,Y 390.087,Z 281.707,A -85,B 0,C 180,E1 -11450.469,E2 -11450.469} C_VEL
LIN {X 0,Y 390.073,Z 281.705,A -85,B 0,C 180,E1 -11453.351,E2 -11453.351} C_VEL
LIN {X 0,Y 390.112,Z 281.705,A -85,B 0,C 180,E1 -11456.767,E2 -11456.767} C_VEL
LIN {X 0,Y 390.037,Z 281.709,A -85,B 0,C 180,E1 -11460.299,E2 -11460.299} C_VEL
LIN {X 0,Y 390.066,Z 281.705,A -85,B 0,C 180,E1 -11464.024,E2 -11464.024} C_VEL
LIN {X 0,Y 390.04,Z 281.712,A -85,B 0,C 180,E1 -11467.55,E2 -11467.55} C_VEL
LIN {X 0,Y 390.052,Z 281.708,A -85,B 0,C 180,E1 -11470.82,E2 -11470.82} C_VEL
LIN {X 0,Y 390.054,Z 281.709,A -85,B 0,C 180,E1 -11473.886,E2 -11473.886} C_VEL
LIN {X 0,Y 390.108,Z 281.7,A -85,B 0,C 180,E1 -11476.796,E2 -11476.796} C_VEL
LIN {X 0,Y 390.071,Z 281.71,A -85,B 0,C 180,E1 -11479.562,E2 -11479.562} C_VEL
LIN {X 0,Y 390.04,Z 281.709,A -85,B 0,C 180,E1 -11482.448,E2 -11482.448} C_VEL
LIN {X 0,Y 390.061,Z 281.711,A -85,B 0,C 180,E1 -11486.044,E2 -11486.044} C_VEL
LIN {X 0,Y 390.044,Z 281.713,A -85,B 0,C 180,E1 -11489.867,E2 -11489.867} C_VEL
LIN {X 0,Y 390.105,Z 281.7,A -85,B 0,C 180,E1 -11493.231,E2 -11493.231} C_VEL
LIN {X 0,Y 390.097,Z 281.703,A -85,B 0,C 180,E1 -11496.75,E2 -11496.75} C_VEL
LIN {X 0,Y 390.094,Z 281.704,A -85,B 0,C 180,E1 -11499.982,E2 -11499.982} C_VEL
LIN {X 0,Y 390.128,Z 281.697,A -85,B 0,C 180,E1 -11503.248,E2 -11503.248} C_VEL
LIN {X 0,Y 390.184,Z 281.697,A -85,B 0,C 180,E1 -11506.561,E2 -11506.561} C_VEL
LIN {X 0,Y 390.194,Z 281.695,A -85,B 0,C 180,E1 -11510.671,E2 -11510.671} C_VEL
LIN {X 0,Y 390.314,Z 281.674,A -85,B 0,C 180,E1 -11513.798,E2 -11513.798} C_VEL
LIN {X 0,Y 390.408,Z 281.662,A -85,B 0,C 180,E1 -11517.937,E2 -11517.937} C_VEL
LIN {X 0,Y 390.537,Z 281.646,A -85,B 0,C 180,E1 -11520,E2 -11520} C_VEL
LIN {X 0,Y 390.298,Z 281.682,A -85,B 0,C 180,E1 -11523.097,E2 -11523.097} C_VEL
LIN {X 0,Y 390.314,Z 281.674,A -85,B 0,C 180,E1 -11526.202,E2 -11526.202} C_VEL
LIN {X 0,Y 390.196,Z 281.695,A -85,B 0,C 180,E1 -11529.329,E2 -11529.329} C_VEL
LIN {X 0,Y 390.167,Z 281.692,A -85,B 0,C 180,E1 -11532.483,E2 -11532.483} C_VEL
LIN {X 0,Y 390.128,Z 281.704,A -85,B 0,C 180,E1 -11535.677,E2 -11535.677} C_VEL
LIN {X 0,Y 390.094,Z 281.701,A -85,B 0,C 180,E1 -11538.922,E2 -11538.922} C_VEL
LIN {X 0,Y 390.027,Z 281.713,A -85,B 0,C 180,E1 -11542.235,E2 -11542.235} C_VEL
LIN {X 0,Y 390.109,Z 281.703,A -85,B 0,C 180,E1 -11545.744,E2 -11545.744} C_VEL
LIN {X 0,Y 390.048,Z 281.707,A -85,B 0,C 180,E1 -11549.11,E2 -11549.11} C_VEL
LIN {X 0,Y 390.034,Z 281.711,A -85,B 0,C 180,E1 -11552.722,E2 -11552.722} C_VEL
LIN {X 0,Y 390.047,Z 281.708,A -85,B 0,C 180,E1 -11555.826,E2 -11555.826} C_VEL
LIN {X 0,Y 390.058,Z 281.706,A -85,B 0,C 180,E1 -11559.218,E2 -11559.218} C_VEL
LIN {X 0,Y 390.035,Z 281.713,A -85,B 0,C 180,E1 -11562.375,E2 -11562.375} C_VEL
LIN {X 0,Y 390.037,Z 281.709,A -85,B 0,C 180,E1 -11565.355,E2 -11565.355} C_VEL
LIN {X 0,Y 390.021,Z 281.711,A -85,B 0,C 180,E1 -11568.187,E2 -11568.187} C_VEL
LIN {X 0,Y 390.082,Z 281.71,A -85,B 0,C 180,E1 -11570.908,E2 -11570.908} C_VEL
LIN {X 0,Y 390.08,Z 281.707,A -85,B 0,C 180,E1 -11574.794,E2 -11574.794} C_VEL
LIN {X 0,Y 390.019,Z 281.711,A -85,B 0,C 180,E1 -11578.496,E2 -11578.496} C_VEL
LIN {X 0,Y 390.034,Z 281.712,A -85,B 0,C 180,E1 -11582.064,E2 -11582.064} C_VEL
LIN {X 0,Y 390.101,Z 281.724,A -85,B 0,C 180,E1 -11584.668,E2 -11584.668} C_VEL
LIN {X 0,Y 391.808,Z 291.59,A -85,B 0,C 180,E1 -11587.316,E2 -11587.316} C_VEL
LIN {X 0,Y 391.735,Z 295.939,A -85,B 0,C 180,E1 -11588.422,E2 -11588.422} C_VEL
LIN {X 0,Y 390.671,Z 312.105,A -85,B 0,C 180,E1 -11592.448,E2 -11592.448} C_VEL
LIN {X 0,Y 390.293,Z 318.884,A -85,B 0,C 180,E1 -11594.087,E2 -11594.087} C_VEL
LIN {X 0,Y 393.5,Z 343.387,A -85,B 0,C 180,E1 -11594.677,E2 -11594.677} C_VEL
LIN {X 0,Y 392.923,Z 395.238,A -85,B 0,C 180,E1 -11595.664,E2 -11595.664} C_VEL
LIN {X 0,Y 392.563,Z 404.312,A -85,B 0,C 180,E1 -11595.948,E2 -11595.948} C_VEL
LIN {X 0,Y 392.203,Z 413.93,A -85,B 0,C 180,E1 -11596.398,E2 -11596.398} C_VEL
LIN {X 0,Y 391.717,Z 424.019,A -85,B 0,C 180,E1 -11597.04,E2 -11597.04} C_VEL
LIN {X 0,Y 391.055,Z 434.501,A -85,B 0,C 180,E1 -11597.941,E2 -11597.941} C_VEL
LIN {X 0,Y 390.555,Z 442.696,A -85,B 0,C 180,E1 -11598.846,E2 -11598.846} C_VEL
LIN {X 0,Y 390.017,Z 450.317,A -85,B 0,C 180,E1 -11599.881,E2 -11599.881} C_VEL
LIN {X 0,Y 389.56,Z 456.586,A -85,B 0,C 180,E1 -11600.918,E2 -11600.918} C_VEL
LIN {X 0,Y 389.255,Z 461.79,A -85,B 0,C 180,E1 -11601.957,E2 -11601.957} C_VEL
LIN {X 0,Y 389.066,Z 466.221,A -85,B 0,C 180,E1 -11603.023,E2 -11603.023} C_VEL
LIN {X 0,Y 388.823,Z 469.918,A -85,B 0,C 180,E1 -11604.104,E2 -11604.104} C_VEL
LIN {X 0,Y 388.793,Z 473.248,A -85,B 0,C 180,E1 -11605.334,E2 -11605.334} C_VEL
LIN {X 0,Y 388.65,Z 476.255,A -85,B 0,C 180,E1 -11606.89,E2 -11606.89} C_VEL
LIN {X 0,Y 388.663,Z 477.598,A -85,B 0,C 180,E1 -11607.927,E2 -11607.927} C_VEL
LIN {X 0,Y 388.701,Z 478.46,A -85,B 0,C 180,E1 -11608.964,E2 -11608.964} C_VEL
LIN {X 0,Y 388.706,Z 478.771,A -85,B 0,C 180,E1 -11610,E2 -11610} C_VEL
LIN {X 0,Y 388.701,Z 478.517,A -85,B 0,C 180,E1 -11611.036,E2 -11611.036} C_VEL
LIN {X 0,Y 388.662,Z 477.796,A -85,B 0,C 180,E1 -11612.072,E2 -11612.072} C_VEL
LIN {X 0,Y 388.649,Z 476.598,A -85,B 0,C 180,E1 -11613.11,E2 -11613.11} C_VEL
LIN {X 0,Y 388.793,Z 473.738,A -85,B 0,C 180,E1 -11614.666,E2 -11614.666} C_VEL
LIN {X 0,Y 388.874,Z 469.611,A -85,B 0,C 180,E1 -11616.225,E2 -11616.225} C_VEL
LIN {X 0,Y 389.201,Z 464.032,A -85,B 0,C 180,E1 -11617.783,E2 -11617.783} C_VEL
LIN {X 0,Y 389.613,Z 457.921,A -85,B 0,C 180,E1 -11619.081,E2 -11619.081} C_VEL
LIN {X 0,Y 390.072,Z 451.966,A -85,B 0,C 180,E1 -11620.117,E2 -11620.117} C_VEL
LIN {X 0,Y 390.65,Z 444.724,A -85,B 0,C 180,E1 -11621.151,E2 -11621.151} C_VEL
LIN {X 0,Y 391.137,Z 436.999,A -85,B 0,C 180,E1 -11622.056,E2 -11622.056} C_VEL
LIN {X 0,Y 391.751,Z 428.887,A -85,B 0,C 180,E1 -11622.827,E2 -11622.827} C_VEL
LIN {X 0,Y 392.275,Z 420.48,A -85,B 0,C 180,E1 -11623.468,E2 -11623.468} C_VEL
LIN {X 0,Y 392.681,Z 411.894,A -85,B 0,C 180,E1 -11623.981,E2 -11623.981} C_VEL
LIN {X 0,Y 393.204,Z 401.659,A -85,B 0,C 180,E1 -11624.425,E2 -11624.425} C_VEL
LIN {X 0,Y 393.572,Z 387.07,A -85,B 0,C 180,E1 -11624.789,E2 -11624.789} C_VEL
LIN {X 0,Y 393.87,Z 341.816,A -85,B 0,C 180,E1 -11625.645,E2 -11625.645} C_VEL
LIN {X 0,Y 390.375,Z 318.073,A -85,B 0,C 180,E1 -11626.27,E2 -11626.27} C_VEL
LIN {X 0,Y 391.186,Z 303.942,A -85,B 0,C 180,E1 -11629.685,E2 -11629.685} C_VEL
LIN {X 0,Y 391.95,Z 292.842,A -85,B 0,C 180,E1 -11632.397,E2 -11632.397} C_VEL
LIN {X 0,Y 390.719,Z 285.021,A -85,B 0,C 180,E1 -11634.437,E2 -11634.437} C_VEL
LIN {X 0,Y 390.09,Z 281.709,A -85,B 0,C 180,E1 -11635.333,E2 -11635.333} C_VEL
LIN {X 0,Y 390.025,Z 281.716,A -85,B 0,C 180,E1 -11639.111,E2 -11639.111} C_VEL
LIN {X 0,Y 390.038,Z 281.715,A -85,B 0,C 180,E1 -11642.721,E2 -11642.721} C_VEL
LIN {X 0,Y 390.05,Z 281.71,A -85,B 0,C 180,E1 -11645.824,E2 -11645.824} C_VEL
LIN {X 0,Y 390.061,Z 281.714,A -85,B 0,C 180,E1 -11649.217,E2 -11649.217} C_VEL
LIN {X 0,Y 390.032,Z 281.712,A -85,B 0,C 180,E1 -11652.373,E2 -11652.373} C_VEL
LIN {X 0,Y 390.037,Z 281.714,A -85,B 0,C 180,E1 -11655.353,E2 -11655.353} C_VEL
LIN {X 0,Y 390.023,Z 281.71,A -85,B 0,C 180,E1 -11658.186,E2 -11658.186} C_VEL
LIN {X 0,Y 390.078,Z 281.706,A -85,B 0,C 180,E1 -11660.906,E2 -11660.906} C_VEL
LIN {X 0,Y 390.076,Z 281.705,A -85,B 0,C 180,E1 -11664.792,E2 -11664.792} C_VEL
LIN {X 0,Y 390.014,Z 281.711,A -85,B 0,C 180,E1 -11668.495,E2 -11668.495} C_VEL
LIN {X 0,Y 390.108,Z 281.696,A -85,B 0,C 180,E1 -11672.069,E2 -11672.069} C_VEL
LIN {X 0,Y 390.066,Z 281.707,A -85,B 0,C 180,E1 -11675.518,E2 -11675.518} C_VEL
LIN {X 0,Y 390.076,Z 281.7,A -85,B 0,C 180,E1 -11679.53,E2 -11679.53} C_VEL
LIN {X 0,Y 390.127,Z 281.693,A -85,B 0,C 180,E1 -11683.248,E2 -11683.248} C_VEL
LIN {X 0,Y 390.183,Z 281.695,A -85,B 0,C 180,E1 -11686.561,E2 -11686.561} C_VEL
LIN {X 0,Y 390.193,Z 281.684,A -85,B 0,C 180,E1 -11690.671,E2 -11690.671} C_VEL
LIN {X 0,Y 390.314,Z 281.673,A -85,B 0,C 180,E1 -11693.798,E2 -11693.798} C_VEL
LIN {X 0,Y 390.405,Z 281.658,A -85,B 0,C 180,E1 -11697.937,E2 -11697.937} C_VEL
LIN {X 0,Y 390.537,Z 281.645,A -85,B 0,C 180,E1 -11700,E2 -11700} C_VEL
LIN {X 0,Y 390.298,Z 281.674,A -85,B 0,C 180,E1 -11703.097,E2 -11703.097} C_VEL
LIN {X 0,Y 390.265,Z 281.677,A -85,B 0,C 180,E1 -11706.492,E2 -11706.492} C_VEL
LIN {X 0,Y 390.192,Z 281.694,A -85,B 0,C 180,E1 -11709.329,E2 -11709.329} C_VEL
LIN {X 0,Y 390.184,Z 281.692,A -85,B 0,C 180,E1 -11713.439,E2 -11713.439} C_VEL
LIN {X 0,Y 390.138,Z 281.697,A -85,B 0,C 180,E1 -11717.308,E2 -11717.308} C_VEL
LIN {X 0,Y 390.077,Z 281.704,A -85,B 0,C 180,E1 -11720.471,E2 -11720.471} C_VEL
LIN {X 0,Y 390.08,Z 281.709,A -85,B 0,C 180,E1 -11723.352,E2 -11723.352} C_VEL
LIN {X 0,Y 390.104,Z 281.701,A -85,B 0,C 180,E1 -11726.769,E2 -11726.769} C_VEL
LIN {X 0,Y 390.035,Z 281.713,A -85,B 0,C 180,E1 -11730.3,E2 -11730.3} C_VEL
LIN {X 0,Y 390.061,Z 281.712,A -85,B 0,C 180,E1 -11734.026,E2 -11734.026} C_VEL
LIN {X 0,Y 390.04,Z 281.712,A -85,B 0,C 180,E1 -11737.552,E2 -11737.552} C_VEL
LIN {X 0,Y 390.081,Z 281.71,A -85,B 0,C 180,E1 -11740.828,E2 -11740.828} C_VEL
LIN {X 0,Y 390.143,Z 281.84,A -85,B 0,C 180,E1 -11741.598,E2 -11741.598} C_VEL
LIN {X 0,Y 391.108,Z 287.245,A -85,B 0,C 180,E1 -11743.066,E2 -11743.066} C_VEL
LIN {X 0,Y 390.743,Z 297.929,A -85,B 0,C 180,E1 -11745.79,E2 -11745.79} C_VEL
LIN {X 0,Y 394.281,Z 316.702,A -85,B 0,C 180,E1 -11746.33,E2 -11746.33} C_VEL
LIN {X 0,Y 393.53,Z 374.569,A -85,B 0,C 180,E1 -11747.438,E2 -11747.438} C_VEL
LIN {X 0,Y 393.2,Z 384.457,A -85,B 0,C 180,E1 -11747.763,E2 -11747.763} C_VEL
LIN {X 0,Y 392.897,Z 395.318,A -85,B 0,C 180,E1 -11748.304,E2 -11748.304} C_VEL
LIN {X 0,Y 392.317,Z 405.418,A -85,B 0,C 180,E1 -11749.009,E2 -11749.009} C_VEL
LIN {X 0,Y 391.696,Z 414.944,A -85,B 0,C 180,E1 -11749.886,E2 -11749.886} C_VEL
LIN {X 0,Y 391.151,Z 422.862,A -85,B 0,C 180,E1 -11750.796,E2 -11750.796} C_VEL
LIN {X 0,Y 390.565,Z 429.94,A -85,B 0,C 180,E1 -11751.79,E2 -11751.79} C_VEL
LIN {X 0,Y 390.106,Z 436.283,A -85,B 0,C 180,E1 -11752.879,E2 -11752.879} C_VEL
LIN {X 0,Y 389.618,Z 442.822,A -85,B 0,C 180,E1 -11754.264,E2 -11754.264} C_VEL
LIN {X 0,Y 389.341,Z 446.852,A -85,B 0,C 180,E1 -11755.348,E2 -11755.348} C_VEL
LIN {X 0,Y 389.028,Z 450.829,A -85,B 0,C 180,E1 -11756.685,E2 -11756.685} C_VEL
LIN {X 0,Y 388.787,Z 454.344,A -85,B 0,C 180,E1 -11758.385,E2 -11758.385} C_VEL
LIN {X 0,Y 388.566,Z 456.615,A -85,B 0,C 180,E1 -11760.248,E2 -11760.248} C_VEL
LIN {X 0,Y 388.481,Z 457.299,A -85,B 0,C 180,E1 -11761.943,E2 -11761.943} C_VEL
LIN {X 0,Y 388.52,Z 456.941,A -85,B 0,C 180,E1 -11763.114,E2 -11763.114} C_VEL
LIN {X 0,Y 388.606,Z 455.411,A -85,B 0,C 180,E1 -11764.724,E2 -11764.724} C_VEL
LIN {X 0,Y 388.8,Z 453.304,A -85,B 0,C 180,E1 -11766.002,E2 -11766.002} C_VEL
LIN {X 0,Y 388.978,Z 450.725,A -85,B 0,C 180,E1 -11767.141,E2 -11767.141} C_VEL
LIN {X 0,Y 389.227,Z 446.436,A -85,B 0,C 180,E1 -11768.554,E2 -11768.554} C_VEL
LIN {X 0,Y 389.563,Z 440.884,A -85,B 0,C 180,E1 -11769.955,E2 -11769.955} C_VEL
LIN {X 0,Y 389.933,Z 435.39,A -85,B 0,C 180,E1 -11771.07,E2 -11771.07} C_VEL
LIN {X 0,Y 390.292,Z 430.522,A -85,B 0,C 180,E1 -11771.904,E2 -11771.904} C_VEL
LIN {X 0,Y 390.72,Z 424.021,A -85,B 0,C 180,E1 -11772.841,E2 -11772.841} C_VEL
LIN {X 0,Y 391.212,Z 416.845,A -85,B 0,C 180,E1 -11773.699,E2 -11773.699} C_VEL
LIN {X 0,Y 391.742,Z 408.376,A -85,B 0,C 180,E1 -11774.522,E2 -11774.522} C_VEL
LIN {X 0,Y 392.21,Z 399.622,A -85,B 0,C 180,E1 -11775.199,E2 -11775.199} C_VEL
LIN {X 0,Y 392.524,Z 390.47,A -85,B 0,C 180,E1 -11775.748,E2 -11775.748} C_VEL
LIN {X 0,Y 392.916,Z 379.355,A -85,B 0,C 180,E1 -11776.225,E2 -11776.225} C_VEL
LIN {X 0,Y 393.18,Z 364.896,A -85,B 0,C 180,E1 -11776.564,E2 -11776.564} C_VEL
LIN {X 0,Y 393.572,Z 315.913,A -85,B 0,C 180,E1 -11777.48,E2 -11777.48} C_VEL
LIN {X 0,Y 390.466,Z 298.224,A -85,B 0,C 180,E1 -11777.956,E2 -11777.956} C_VEL
LIN {X 0,Y 390.916,Z 288.498,A -85,B 0,C 180,E1 -11780.689,E2 -11780.689} C_VEL
LIN {X 0,Y 390.556,Z 283.141,A -85,B 0,C 180,E1 -11782.244,E2 -11782.244} C_VEL
LIN {X 0,Y 390.307,Z 281.681,A -85,B 0,C 180,E1 -11782.759,E2 -11782.759} C_VEL
LIN {X 0,Y 390.226,Z 281.686,A -85,B 0,C 180,E1 -11784.834,E2 -11784.834} C_VEL
LIN {X 0,Y 390.42,Z 281.667,A -85,B 0,C 180,E1 -11787.937,E2 -11787.937} C_VEL
LIN {X 0,Y 390.441,Z 281.659,A -85,B 0,C 180,E1 -11790.479,E2 -11790.479} C_VEL
LIN {X 0,Y 389.624,Z 281.762,A -85,B 0,C 180,E1 -11791.339,E2 -11791.339} C_VEL
LIN {X 0,Y 386.603,Z 282.137,A -85,B 0,C 180,E1 -11792.735,E2 -11792.735} C_VEL
LIN {X 0,Y 384.168,Z 282.444,A -85,B 0,C 180,E1 -11793.863,E2 -11793.863} C_VEL
LIN {X 0,Y 383.198,Z 282.561,A -85,B 0,C 180,E1 -11794.737,E2 -11794.737} C_VEL
LIN {X 0,Y 383.156,Z 282.565,A -85,B 0,C 180,E1 -11795.033,E2 -11795.033} C_VEL
LIN {X 0,Y 383.218,Z 282.558,A -85,B 0,C 180,E1 -11797.376,E2 -11797.376} C_VEL
LIN {X 0,Y 383.132,Z 282.572,A -85,B 0,C 180,E1 -11800.57,E2 -11800.57} C_VEL
LIN {X 0,Y 383.128,Z 282.57,A -85,B 0,C 180,E1 -11803.796,E2 -11803.796} C_VEL
LIN {X 0,Y 383.076,Z 282.575,A -85,B 0,C 180,E1 -11807.445,E2 -11807.445} C_VEL
LIN {X 0,Y 383.029,Z 282.589,A -85,B 0,C 180,E1 -11810.646,E2 -11810.646} C_VEL
LIN {X 0,Y 383.025,Z 282.582,A -85,B 0,C 180,E1 -11813.807,E2 -11813.807} C_VEL
LIN {X 0,Y 383.079,Z 282.576,A -85,B 0,C 180,E1 -11816.123,E2 -11816.123} C_VEL
LIN {X 0,Y 382.99,Z 282.587,A -85,B 0,C 180,E1 -11819.699,E2 -11819.699} C_VEL
LIN {X 0,Y 383,Z 282.589,A -85,B 0,C 180,E1 -11823.4,E2 -11823.4} C_VEL
LIN {X 0,Y 383.028,Z 282.581,A -85,B 0,C 180,E1 -11826.163,E2 -11826.163} C_VEL
LIN {X 0,Y 383.005,Z 282.585,A -85,B 0,C 180,E1 -11829.957,E2 -11829.957} C_VEL
LIN {X 0,Y 383.001,Z 282.586,A -85,B 0,C 180,E1 -11832.778,E2 -11832.778} C_VEL
LIN {X 0,Y 383.032,Z 282.585,A -85,B 0,C 180,E1 -11835.794,E2 -11835.794} C_VEL
LIN {X 0,Y 383.038,Z 282.58,A -85,B 0,C 180,E1 -11838.785,E2 -11838.785} C_VEL
LIN {X 0,Y 382.996,Z 282.589,A -85,B 0,C 180,E1 -11842.095,E2 -11842.095} C_VEL
LIN {X 0,Y 383.011,Z 282.585,A -85,B 0,C 180,E1 -11845.331,E2 -11845.331} C_VEL
LIN {X 0,Y 382.978,Z 282.588,A -85,B 0,C 180,E1 -11849.081,E2 -11849.081} C_VEL
LIN {X 0,Y 383.048,Z 282.58,A -85,B 0,C 180,E1 -11852.697,E2 -11852.697} C_VEL
LIN {X 0,Y 383.043,Z 282.58,A -85,B 0,C 180,E1 -11855.039,E2 -11855.039} C_VEL
LIN {X 0,Y 382.983,Z 282.593,A -85,B 0,C 180,E1 -11858.468,E2 -11858.468} C_VEL
LIN {X 0,Y 383.052,Z 282.579,A -85,B 0,C 180,E1 -11861.826,E2 -11861.826} C_VEL
LIN {X 0,Y 383.099,Z 282.574,A -85,B 0,C 180,E1 -11865.118,E2 -11865.118} C_VEL
LIN {X 0,Y 383.086,Z 282.578,A -85,B 0,C 180,E1 -11868.357,E2 -11868.357} C_VEL
LIN {X 0,Y 383.254,Z 282.553,A -85,B 0,C 180,E1 -11871.975,E2 -11871.975} C_VEL
LIN {X 0,Y 383.186,Z 282.567,A -85,B 0,C 180,E1 -11874.738,E2 -11874.738} C_VEL
LIN {X 0,Y 383.376,Z 282.538,A -85,B 0,C 180,E1 -11877.899,E2 -11877.899} C_VEL
LIN {X 0,Y 383.507,Z 282.522,A -85,B 0,C 180,E1 -11880,E2 -11880} C_VEL
LIN {X 0,Y 383.235,Z 282.562,A -85,B 0,C 180,E1 -11883.154,E2 -11883.154} C_VEL
LIN {X 0,Y 383.27,Z 282.551,A -85,B 0,C 180,E1 -11886.316,E2 -11886.316} C_VEL
LIN {X 0,Y 383.143,Z 282.574,A -85,B 0,C 180,E1 -11889.502,E2 -11889.502} C_VEL
LIN {X 0,Y 383.131,Z 282.569,A -85,B 0,C 180,E1 -11892.716,E2 -11892.716} C_VEL
LIN {X 0,Y 383.07,Z 282.58,A -85,B 0,C 180,E1 -11895.974,E2 -11895.974} C_VEL
LIN {X 0,Y 383.049,Z 282.581,A -85,B 0,C 180,E1 -11899.284,E2 -11899.284} C_VEL
LIN {X 0,Y 382.984,Z 282.587,A -85,B 0,C 180,E1 -11902.666,E2 -11902.666} C_VEL
LIN {X 0,Y 383.07,Z 282.582,A -85,B 0,C 180,E1 -11906.124,E2 -11906.124} C_VEL
LIN {X 0,Y 382.982,Z 282.589,A -85,B 0,C 180,E1 -11909.701,E2 -11909.701} C_VEL
LIN {X 0,Y 382.995,Z 282.586,A -85,B 0,C 180,E1 -11913.401,E2 -11913.401} C_VEL
LIN {X 0,Y 383.023,Z 282.587,A -85,B 0,C 180,E1 -11916.165,E2 -11916.165} C_VEL
LIN {X 0,Y 383,Z 282.586,A -85,B 0,C 180,E1 -11919.959,E2 -11919.959} C_VEL
LIN {X 0,Y 382.999,Z 282.59,A -85,B 0,C 180,E1 -11922.779,E2 -11922.779} C_VEL
LIN {X 0,Y 382.99,Z 282.586,A -85,B 0,C 180,E1 -11925.79,E2 -11925.79} C_VEL
LIN {X 0,Y 382.98,Z 282.594,A -85,B 0,C 180,E1 -11928.797,E2 -11928.797} C_VEL
LIN {X 0,Y 382.993,Z 282.586,A -85,B 0,C 180,E1 -11932.097,E2 -11932.097} C_VEL
LIN {X 0,Y 383.013,Z 282.587,A -85,B 0,C 180,E1 -11935.333,E2 -11935.333} C_VEL
LIN {X 0,Y 382.978,Z 282.594,A -85,B 0,C 180,E1 -11939.082,E2 -11939.082} C_VEL
LIN {X 0,Y 382.989,Z 282.591,A -85,B 0,C 180,E1 -11942.694,E2 -11942.694} C_VEL
LIN {X 0,Y 383.041,Z 282.672,A -85,B 0,C 180,E1 -11944.498,E2 -11944.498} C_VEL
LIN {X 0,Y 384.794,Z 292.397,A -85,B 0,C 180,E1 -11947.163,E2 -11947.163} C_VEL
LIN {X 0,Y 384.742,Z 296.745,A -85,B 0,C 180,E1 -11948.291,E2 -11948.291} C_VEL
LIN {X 0,Y 383.644,Z 312.496,A -85,B 0,C 180,E1 -11952.286,E2 -11952.286} C_VEL
LIN {X 0,Y 383.299,Z 318.765,A -85,B 0,C 180,E1 -11953.814,E2 -11953.814} C_VEL
LIN {X 0,Y 386.605,Z 344.536,A -85,B 0,C 180,E1 -11954.446,E2 -11954.446} C_VEL
LIN {X 0,Y 386.023,Z 395.399,A -85,B 0,C 180,E1 -11955.436,E2 -11955.436} C_VEL
LIN {X 0,Y 385.627,Z 405.171,A -85,B 0,C 180,E1 -11955.757,E2 -11955.757} C_VEL
LIN {X 0,Y 385.091,Z 416.849,A -85,B 0,C 180,E1 -11956.343,E2 -11956.343} C_VEL
LIN {X 0,Y 384.557,Z 426.81,A -85,B 0,C 180,E1 -11957.064,E2 -11957.064} C_VEL
LIN {X 0,Y 384.02,Z 435.317,A -85,B 0,C 180,E1 -11957.851,E2 -11957.851} C_VEL
LIN {X 0,Y 383.52,Z 443.342,A -85,B 0,C 180,E1 -11958.773,E2 -11958.773} C_VEL
LIN {X 0,Y 383.003,Z 449.967,A -85,B 0,C 180,E1 -11959.694,E2 -11959.694} C_VEL
LIN {X 0,Y 382.54,Z 456.263,A -85,B 0,C 180,E1 -11960.75,E2 -11960.75} C_VEL
LIN {X 0,Y 382.185,Z 461.489,A -85,B 0,C 180,E1 -11961.807,E2 -11961.807} C_VEL
LIN {X 0,Y 381.936,Z 466.806,A -85,B 0,C 180,E1 -11963.131,E2 -11963.131} C_VEL
LIN {X 0,Y 381.719,Z 470.138,A -85,B 0,C 180,E1 -11964.161,E2 -11964.161} C_VEL
LIN {X 0,Y 381.705,Z 473.002,A -85,B 0,C 180,E1 -11965.247,E2 -11965.247} C_VEL
LIN {X 0,Y 381.562,Z 476.025,A -85,B 0,C 180,E1 -11966.832,E2 -11966.832} C_VEL
LIN {X 0,Y 381.563,Z 477.382,A -85,B 0,C 180,E1 -11967.889,E2 -11967.889} C_VEL
LIN {X 0,Y 381.601,Z 478.256,A -85,B 0,C 180,E1 -11968.945,E2 -11968.945} C_VEL
LIN {X 0,Y 381.637,Z 478.57,A -85,B 0,C 180,E1 -11970,E2 -11970} C_VEL
LIN {X 0,Y 381.601,Z 478.327,A -85,B 0,C 180,E1 -11971.055,E2 -11971.055} C_VEL
LIN {X 0,Y 381.561,Z 477.617,A -85,B 0,C 180,E1 -11972.111,E2 -11972.111} C_VEL
LIN {X 0,Y 381.561,Z 476.432,A -85,B 0,C 180,E1 -11973.168,E2 -11973.168} C_VEL
LIN {X 0,Y 381.669,Z 474.739,A -85,B 0,C 180,E1 -11974.224,E2 -11974.224} C_VEL
LIN {X 0,Y 381.729,Z 470.888,A -85,B 0,C 180,E1 -11975.852,E2 -11975.852} C_VEL
LIN {X 0,Y 381.997,Z 467.818,A -85,B 0,C 180,E1 -11976.868,E2 -11976.868} C_VEL
LIN {X 0,Y 382.228,Z 462.753,A -85,B 0,C 180,E1 -11978.192,E2 -11978.192} C_VEL
LIN {X 0,Y 382.589,Z 457.825,A -85,B 0,C 180,E1 -11979.249,E2 -11979.249} C_VEL
LIN {X 0,Y 383.078,Z 451.89,A -85,B 0,C 180,E1 -11980.304,E2 -11980.304} C_VEL
LIN {X 0,Y 383.681,Z 444.671,A -85,B 0,C 180,E1 -11981.356,E2 -11981.356} C_VEL
LIN {X 0,Y 384.21,Z 436.975,A -85,B 0,C 180,E1 -11982.277,E2 -11982.277} C_VEL
LIN {X 0,Y 384.838,Z 428.901,A -85,B 0,C 180,E1 -11983.061,E2 -11983.061} C_VEL
LIN {X 0,Y 385.392,Z 420.547,A -85,B 0,C 180,E1 -11983.713,E2 -11983.713} C_VEL
LIN {X 0,Y 385.816,Z 412.039,A -85,B 0,C 180,E1 -11984.235,E2 -11984.235} C_VEL
LIN {X 0,Y 386.349,Z 401.94,A -85,B 0,C 180,E1 -11984.686,E2 -11984.686} C_VEL
LIN {X 0,Y 386.709,Z 389.838,A -85,B 0,C 180,E1 -11985.021,E2 -11985.021} C_VEL
LIN {X 0,Y 387.16,Z 343.255,A -85,B 0,C 180,E1 -11985.914,E2 -11985.914} C_VEL
LIN {X 0,Y 383.643,Z 319.441,A -85,B 0,C 180,E1 -11986.551,E2 -11986.551} C_VEL
LIN {X 0,Y 383.434,Z 317.821,A -85,B 0,C 180,E1 -11986.607,E2 -11986.607} C_VEL
LIN {X 0,Y 384.208,Z 304.934,A -85,B 0,C 180,E1 -11989.779,E2 -11989.779} C_VEL
LIN {X 0,Y 384.989,Z 293.841,A -85,B 0,C 180,E1 -11992.541,E2 -11992.541} C_VEL
LIN {X 0,Y 383.506,Z 284.919,A -85,B 0,C 180,E1 -11994.928,E2 -11994.928} C_VEL
LIN {X 0,Y 383.024,Z 282.588,A -85,B 0,C 180,E1 -11995.615,E2 -11995.615} C_VEL
LIN {X 0,Y 382.977,Z 282.596,A -85,B 0,C 180,E1 -11998.497,E2 -11998.497} C_VEL
LIN {X 0,Y 383.005,Z 282.587,A -85,B 0,C 180,E1 -12002.149,E2 -12002.149} C_VEL
LIN {X 0,Y 383.013,Z 282.59,A -85,B 0,C 180,E1 -12004.667,E2 -12004.667} C_VEL
LIN {X 0,Y 382.993,Z 282.592,A -85,B 0,C 180,E1 -12007.903,E2 -12007.903} C_VEL
LIN {X 0,Y 382.975,Z 282.596,A -85,B 0,C 180,E1 -12011.347,E2 -12011.347} C_VEL
LIN {X 0,Y 382.988,Z 282.592,A -85,B 0,C 180,E1 -12014.302,E2 -12014.302} C_VEL
LIN {X 0,Y 383.003,Z 282.593,A -85,B 0,C 180,E1 -12017.239,E2 -12017.239} C_VEL
LIN {X 0,Y 383.005,Z 282.586,A -85,B 0,C 180,E1 -12020.413,E2 -12020.413} C_VEL
LIN {X 0,Y 383.016,Z 282.587,A -85,B 0,C 180,E1 -12024.044,E2 -12024.044} C_VEL
LIN {X 0,Y 382.977,Z 282.586,A -85,B 0,C 180,E1 -12027.577,E2 -12027.577} C_VEL
LIN {X 0,Y 382.982,Z 282.589,A -85,B 0,C 180,E1 -12030.299,E2 -12030.299} C_VEL
LIN {X 0,Y 383.07,Z 282.577,A -85,B 0,C 180,E1 -12034.02,E2 -12034.02} C_VEL
LIN {X 0,Y 382.98,Z 282.585,A -85,B 0,C 180,E1 -12037.334,E2 -12037.334} C_VEL
LIN {X 0,Y 383.049,Z 282.582,A -85,B 0,C 180,E1 -12040.716,E2 -12040.716} C_VEL
LIN {X 0,Y 383.069,Z 282.573,A -85,B 0,C 180,E1 -12044.026,E2 -12044.026} C_VEL
LIN {X 0,Y 383.125,Z 282.57,A -85,B 0,C 180,E1 -12047.284,E2 -12047.284} C_VEL
LIN {X 0,Y 383.14,Z 282.562,A -85,B 0,C 180,E1 -12050.498,E2 -12050.498} C_VEL
LIN {X 0,Y 383.271,Z 282.551,A -85,B 0,C 180,E1 -12053.684,E2 -12053.684} C_VEL
LIN {X 0,Y 383.372,Z 282.534,A -85,B 0,C 180,E1 -12057.899,E2 -12057.899} C_VEL
LIN {X 0,Y 383.506,Z 282.521,A -85,B 0,C 180,E1 -12060,E2 -12060} C_VEL
LIN {X 0,Y 383.234,Z 282.554,A -85,B 0,C 180,E1 -12063.154,E2 -12063.154} C_VEL
LIN {X 0,Y 383.228,Z 282.555,A -85,B 0,C 180,E1 -12066.48,E2 -12066.48} C_VEL
LIN {X 0,Y 383.139,Z 282.574,A -85,B 0,C 180,E1 -12069.503,E2 -12069.503} C_VEL
LIN {X 0,Y 383.115,Z 282.574,A -85,B 0,C 180,E1 -12073.537,E2 -12073.537} C_VEL
LIN {X 0,Y 383.084,Z 282.577,A -85,B 0,C 180,E1 -12077.455,E2 -12077.455} C_VEL
LIN {X 0,Y 383.018,Z 282.583,A -85,B 0,C 180,E1 -12080.647,E2 -12080.647} C_VEL
LIN {X 0,Y 383.024,Z 282.588,A -85,B 0,C 180,E1 -12083.808,E2 -12083.808} C_VEL
LIN {X 0,Y 383.071,Z 282.58,A -85,B 0,C 180,E1 -12086.124,E2 -12086.124} C_VEL
LIN {X 0,Y 383.041,Z 282.582,A -85,B 0,C 180,E1 -12088.493,E2 -12088.493} C_VEL
LIN {X 0,Y 383.003,Z 282.592,A -85,B 0,C 180,E1 -12092.15,E2 -12092.15} C_VEL
LIN {X 0,Y 383.011,Z 282.584,A -85,B 0,C 180,E1 -12094.669,E2 -12094.669} C_VEL
LIN {X 0,Y 382.996,Z 282.592,A -85,B 0,C 180,E1 -12097.905,E2 -12097.905} C_VEL
LIN {X 0,Y 383.074,Z 282.621,A -85,B 0,C 180,E1 -12101.336,E2 -12101.336} C_VEL
LIN {X 0,Y 384.157,Z 288.508,A -85,B 0,C 180,E1 -12102.966,E2 -12102.966} C_VEL
LIN {X 0,Y 383.809,Z 298.111,A -85,B 0,C 180,E1 -12105.46,E2 -12105.46} C_VEL
LIN {X 0,Y 387.501,Z 318.018,A -85,B 0,C 180,E1 -12106.044,E2 -12106.044} C_VEL
LIN {X 0,Y 386.687,Z 375.413,A -85,B 0,C 180,E1 -12107.169,E2 -12107.169} C_VEL
LIN {X 0,Y 386.372,Z 385.656,A -85,B 0,C 180,E1 -12107.525,E2 -12107.525} C_VEL
LIN {X 0,Y 385.914,Z 397.348,A -85,B 0,C 180,E1 -12108.15,E2 -12108.15} C_VEL
LIN {X 0,Y 385.383,Z 406.612,A -85,B 0,C 180,E1 -12108.84,E2 -12108.84} C_VEL
LIN {X 0,Y 384.843,Z 414.612,A -85,B 0,C 180,E1 -12109.589,E2 -12109.589} C_VEL
LIN {X 0,Y 384.309,Z 421.552,A -85,B 0,C 180,E1 -12110.376,E2 -12110.376} C_VEL
LIN {X 0,Y 383.738,Z 428.449,A -85,B 0,C 180,E1 -12111.32,E2 -12111.32} C_VEL
LIN {X 0,Y 383.256,Z 434.854,A -85,B 0,C 180,E1 -12112.387,E2 -12112.387} C_VEL
LIN {X 0,Y 382.856,Z 439.813,A -85,B 0,C 180,E1 -12113.374,E2 -12113.374} C_VEL
LIN {X 0,Y 382.462,Z 444.989,A -85,B 0,C 180,E1 -12114.633,E2 -12114.633} C_VEL
LIN {X 0,Y 382.062,Z 449.065,A -85,B 0,C 180,E1 -12115.871,E2 -12115.871} C_VEL
LIN {X 0,Y 381.93,Z 452.27,A -85,B 0,C 180,E1 -12117.124,E2 -12117.124} C_VEL
LIN {X 0,Y 381.829,Z 453.83,A -85,B 0,C 180,E1 -12117.853,E2 -12117.853} C_VEL
LIN {X 0,Y 381.62,Z 455.552,A -85,B 0,C 180,E1 -12118.96,E2 -12118.96} C_VEL
LIN {X 0,Y 381.482,Z 456.793,A -85,B 0,C 180,E1 -12120.172,E2 -12120.172} C_VEL
LIN {X 0,Y 381.408,Z 457.431,A -85,B 0,C 180,E1 -12122.187,E2 -12122.187} C_VEL
LIN {X 0,Y 381.442,Z 456.627,A -85,B 0,C 180,E1 -12123.757,E2 -12123.757} C_VEL
LIN {X 0,Y 381.531,Z 455.326,A -85,B 0,C 180,E1 -12124.934,E2 -12124.934} C_VEL
LIN {X 0,Y 381.721,Z 453.384,A -85,B 0,C 180,E1 -12126.107,E2 -12126.107} C_VEL
LIN {X 0,Y 381.905,Z 450.779,A -85,B 0,C 180,E1 -12127.267,E2 -12127.267} C_VEL
LIN {X 0,Y 382.174,Z 446.44,A -85,B 0,C 180,E1 -12128.704,E2 -12128.704} C_VEL
LIN {X 0,Y 382.452,Z 442.019,A -85,B 0,C 180,E1 -12129.867,E2 -12129.867} C_VEL
LIN {X 0,Y 382.847,Z 436.817,A -85,B 0,C 180,E1 -12130.984,E2 -12130.984} C_VEL
LIN {X 0,Y 383.336,Z 430.008,A -85,B 0,C 180,E1 -12132.171,E2 -12132.171} C_VEL
LIN {X 0,Y 383.781,Z 423.562,A -85,B 0,C 180,E1 -12133.1,E2 -12133.1} C_VEL
LIN {X 0,Y 384.26,Z 416.552,A -85,B 0,C 180,E1 -12133.941,E2 -12133.941} C_VEL
LIN {X 0,Y 384.841,Z 407.939,A -85,B 0,C 180,E1 -12134.781,E2 -12134.781} C_VEL
LIN {X 0,Y 385.334,Z 397.989,A -85,B 0,C 180,E1 -12135.544,E2 -12135.544} C_VEL
LIN {X 0,Y 385.796,Z 386.12,A -85,B 0,C 180,E1 -12136.201,E2 -12136.201} C_VEL
LIN {X 0,Y 386.101,Z 375.277,A -85,B 0,C 180,E1 -12136.581,E2 -12136.581} C_VEL
LIN {X 0,Y 386.802,Z 317.508,A -85,B 0,C 180,E1 -12137.707,E2 -12137.707} C_VEL
LIN {X 0,Y 383.48,Z 298.372,A -85,B 0,C 180,E1 -12138.236,E2 -12138.236} C_VEL
LIN {X 0,Y 383.917,Z 288.548,A -85,B 0,C 180,E1 -12141.049,E2 -12141.049} C_VEL
LIN {X 0,Y 383.278,Z 282.557,A -85,B 0,C 180,E1 -12142.857,E2 -12142.857} C_VEL
LIN {X 0,Y 383.248,Z 282.554,A -85,B 0,C 180,E1 -12146.846,E2 -12146.846} C_VEL
LIN {X 0,Y 383.52,Z 282.527,A -85,B 0,C 180,E1 -12150,E2 -12150} C_VEL
LIN {X 0,Y 383.248,Z 282.554,A -85,B 0,C 180,E1 -12153.154,E2 -12153.154} C_VEL
LIN {X 0,Y 383.156,Z 282.565,A -85,B 0,C 180,E1 -12155.033,E2 -12155.033} C_VEL
LIN {X 0,Y 382.594,Z 282.641,A -85,B 0,C 180,E1 -12155.911,E2 -12155.911} C_VEL
LIN {X 0,Y 379.79,Z 282.99,A -85,B 0,C 180,E1 -12157.34,E2 -12157.34} C_VEL
LIN {X 0,Y 377.328,Z 283.298,A -85,B 0,C 180,E1 -12158.495,E2 -12158.495} C_VEL
LIN {X 0,Y 376.228,Z 283.432,A -85,B 0,C 180,E1 -12159.388,E2 -12159.388} C_VEL
LIN {X 0,Y 376.119,Z 283.443,A -85,B 0,C 180,E1 -12159.691,E2 -12159.691} C_VEL
LIN {X 0,Y 376.091,Z 283.446,A -85,B 0,C 180,E1 -12163.657,E2 -12163.657} C_VEL
LIN {X 0,Y 376.033,Z 283.453,A -85,B 0,C 180,E1 -12167.399,E2 -12167.399} C_VEL
LIN {X 0,Y 375.978,Z 283.465,A -85,B 0,C 180,E1 -12170.831,E2 -12170.831} C_VEL
LIN {X 0,Y 375.989,Z 283.46,A -85,B 0,C 180,E1 -12174.281,E2 -12174.281} C_VEL
LIN {X 0,Y 376.019,Z 283.459,A -85,B 0,C 180,E1 -12176.651,E2 -12176.651} C_VEL
LIN {X 0,Y 375.963,Z 283.462,A -85,B 0,C 180,E1 -12180.312,E2 -12180.312} C_VEL
LIN {X 0,Y 375.957,Z 283.462,A -85,B 0,C 180,E1 -12184.111,E2 -12184.111} C_VEL
LIN {X 0,Y 375.95,Z 283.465,A -85,B 0,C 180,E1 -12186.74,E2 -12186.74} C_VEL
LIN {X 0,Y 375.985,Z 283.46,A -85,B 0,C 180,E1 -12189.97,E2 -12189.97} C_VEL
LIN {X 0,Y 375.932,Z 283.469,A -85,B 0,C 180,E1 -12193.764,E2 -12193.764} C_VEL
LIN {X 0,Y 375.983,Z 283.459,A -85,B 0,C 180,E1 -12196.801,E2 -12196.801} C_VEL
LIN {X 0,Y 375.993,Z 283.461,A -85,B 0,C 180,E1 -12200.027,E2 -12200.027} C_VEL
LIN {X 0,Y 375.958,Z 283.466,A -85,B 0,C 180,E1 -12203.494,E2 -12203.494} C_VEL
LIN {X 0,Y 375.953,Z 283.47,A -85,B 0,C 180,E1 -12205.888,E2 -12205.888} C_VEL
LIN {X 0,Y 375.96,Z 283.465,A -85,B 0,C 180,E1 -12209.687,E2 -12209.687} C_VEL
LIN {X 0,Y 375.995,Z 283.465,A -85,B 0,C 180,E1 -12212.141,E2 -12212.141} C_VEL
LIN {X 0,Y 375.997,Z 283.461,A -85,B 0,C 180,E1 -12214.538,E2 -12214.538} C_VEL
LIN {X 0,Y 375.953,Z 283.467,A -85,B 0,C 180,E1 -12218.045,E2 -12218.045} C_VEL
LIN {X 0,Y 375.999,Z 283.457,A -85,B 0,C 180,E1 -12221.473,E2 -12221.473} C_VEL
LIN {X 0,Y 376.048,Z 283.455,A -85,B 0,C 180,E1 -12224.832,E2 -12224.832} C_VEL
LIN {X 0,Y 376.039,Z 283.454,A -85,B 0,C 180,E1 -12228.136,E2 -12228.136} C_VEL
LIN {X 0,Y 376.209,Z 283.431,A -85,B 0,C 180,E1 -12231.918,E2 -12231.918} C_VEL
LIN {X 0,Y 376.158,Z 283.441,A -85,B 0,C 180,E1 -12234.64,E2 -12234.64} C_VEL
LIN {X 0,Y 376.342,Z 283.414,A -85,B 0,C 180,E1 -12237.859,E2 -12237.859} C_VEL
LIN {X 0,Y 376.477,Z 283.398,A -85,B 0,C 180,E1 -12240,E2 -12240} C_VEL
LIN {X 0,Y 376.174,Z 283.443,A -85,B 0,C 180,E1 -12243.213,E2 -12243.213} C_VEL
LIN {X 0,Y 376.228,Z 283.428,A -85,B 0,C 180,E1 -12246.435,E2 -12246.435} C_VEL
LIN {X 0,Y 376.111,Z 283.448,A -85,B 0,C 180,E1 -12249.682,E2 -12249.682} C_VEL
LIN {X 0,Y 376.079,Z 283.454,A -85,B 0,C 180,E1 -12253.658,E2 -12253.658} C_VEL
LIN {X 0,Y 376.033,Z 283.459,A -85,B 0,C 180,E1 -12257.607,E2 -12257.607} C_VEL
LIN {X 0,Y 375.968,Z 283.461,A -85,B 0,C 180,E1 -12260.833,E2 -12260.833} C_VEL
LIN {X 0,Y 375.979,Z 283.463,A -85,B 0,C 180,E1 -12264.282,E2 -12264.282} C_VEL
LIN {X 0,Y 376.01,Z 283.457,A -85,B 0,C 180,E1 -12266.653,E2 -12266.653} C_VEL
LIN {X 0,Y 375.955,Z 283.468,A -85,B 0,C 180,E1 -12270.313,E2 -12270.313} C_VEL
LIN {X 0,Y 375.951,Z 283.468,A -85,B 0,C 180,E1 -12274.112,E2 -12274.112} C_VEL
LIN {X 0,Y 375.945,Z 283.467,A -85,B 0,C 180,E1 -12276.742,E2 -12276.742} C_VEL
LIN {X 0,Y 375.98,Z 283.461,A -85,B 0,C 180,E1 -12279.971,E2 -12279.971} C_VEL
LIN {X 0,Y 375.922,Z 283.467,A -85,B 0,C 180,E1 -12283.767,E2 -12283.767} C_VEL
LIN {X 0,Y 375.928,Z 283.473,A -85,B 0,C 180,E1 -12286.811,E2 -12286.811} C_VEL
LIN {X 0,Y 375.956,Z 283.466,A -85,B 0,C 180,E1 -12290.538,E2 -12290.538} C_VEL
LIN {X 0,Y 375.959,Z 283.464,A -85,B 0,C 180,E1 -12293.497,E2 -12293.497} C_VEL
LIN {X 0,Y 375.956,Z 283.463,A -85,B 0,C 180,E1 -12295.889,E2 -12295.889} C_VEL
LIN {X 0,Y 375.959,Z 283.464,A -85,B 0,C 180,E1 -12299.688,E2 -12299.688} C_VEL
LIN {X 0,Y 375.931,Z 283.469,A -85,B 0,C 180,E1 -12302.137,E2 -12302.137} C_VEL
LIN {X 0,Y 376.005,Z 283.576,A -85,B 0,C 180,E1 -12304.315,E2 -12304.315} C_VEL
LIN {X 0,Y 377.773,Z 293.194,A -85,B 0,C 180,E1 -12307.004,E2 -12307.004} C_VEL
LIN {X 0,Y 377.76,Z 297.545,A -85,B 0,C 180,E1 -12308.156,E2 -12308.156} C_VEL
LIN {X 0,Y 376.589,Z 313.485,A -85,B 0,C 180,E1 -12312.275,E2 -12312.275} C_VEL
LIN {X 0,Y 376.281,Z 318.346,A -85,B 0,C 180,E1 -12313.521,E2 -12313.521} C_VEL
LIN {X 0,Y 379.744,Z 345.606,A -85,B 0,C 180,E1 -12314.206,E2 -12314.206} C_VEL
LIN {X 0,Y 379.106,Z 395.552,A -85,B 0,C 180,E1 -12315.198,E2 -12315.198} C_VEL
LIN {X 0,Y 378.71,Z 405.2,A -85,B 0,C 180,E1 -12315.526,E2 -12315.526} C_VEL
LIN {X 0,Y 378.169,Z 416.255,A -85,B 0,C 180,E1 -12316.088,E2 -12316.088} C_VEL
LIN {X 0,Y 377.635,Z 426.342,A -85,B 0,C 180,E1 -12316.822,E2 -12316.822} C_VEL
LIN {X 0,Y 377.06,Z 434.897,A -85,B 0,C 180,E1 -12317.623,E2 -12317.623} C_VEL
LIN {X 0,Y 376.505,Z 442.959,A -85,B 0,C 180,E1 -12318.561,E2 -12318.561} C_VEL
LIN {X 0,Y 376.003,Z 449.618,A -85,B 0,C 180,E1 -12319.5,E2 -12319.5} C_VEL
LIN {X 0,Y 375.534,Z 455.941,A -85,B 0,C 180,E1 -12320.575,E2 -12320.575} C_VEL
LIN {X 0,Y 375.139,Z 461.189,A -85,B 0,C 180,E1 -12321.652,E2 -12321.652} C_VEL
LIN {X 0,Y 374.874,Z 466.526,A -85,B 0,C 180,E1 -12323.001,E2 -12323.001} C_VEL
LIN {X 0,Y 374.616,Z 470.352,A -85,B 0,C 180,E1 -12324.218,E2 -12324.218} C_VEL
LIN {X 0,Y 374.6,Z 473.917,A -85,B 0,C 180,E1 -12325.696,E2 -12325.696} C_VEL
LIN {X 0,Y 374.478,Z 475.794,A -85,B 0,C 180,E1 -12326.772,E2 -12326.772} C_VEL
LIN {X 0,Y 374.463,Z 477.165,A -85,B 0,C 180,E1 -12327.849,E2 -12327.849} C_VEL
LIN {X 0,Y 374.501,Z 478.051,A -85,B 0,C 180,E1 -12328.925,E2 -12328.925} C_VEL
LIN {X 0,Y 374.552,Z 478.367,A -85,B 0,C 180,E1 -12330,E2 -12330} C_VEL
LIN {X 0,Y 374.501,Z 478.135,A -85,B 0,C 180,E1 -12331.075,E2 -12331.075} C_VEL
LIN {X 0,Y 374.46,Z 477.439,A -85,B 0,C 180,E1 -12332.151,E2 -12332.151} C_VEL
LIN {X 0,Y 374.476,Z 476.266,A -85,B 0,C 180,E1 -12333.227,E2 -12333.227} C_VEL
LIN {X 0,Y 374.6,Z 474.581,A -85,B 0,C 180,E1 -12334.304,E2 -12334.304} C_VEL
LIN {X 0,Y 374.629,Z 471.214,A -85,B 0,C 180,E1 -12335.799,E2 -12335.799} C_VEL
LIN {X 0,Y 374.942,Z 467.691,A -85,B 0,C 180,E1 -12336.998,E2 -12336.998} C_VEL
LIN {X 0,Y 375.175,Z 462.64,A -85,B 0,C 180,E1 -12338.347,E2 -12338.347} C_VEL
LIN {X 0,Y 375.705,Z 456.307,A -85,B 0,C 180,E1 -12339.692,E2 -12339.692} C_VEL
LIN {X 0,Y 376.23,Z 450.115,A -85,B 0,C 180,E1 -12340.766,E2 -12340.766} C_VEL
LIN {X 0,Y 376.791,Z 443.615,A -85,B 0,C 180,E1 -12341.703,E2 -12341.703} C_VEL
LIN {X 0,Y 377.403,Z 435.754,A -85,B 0,C 180,E1 -12342.639,E2 -12342.639} C_VEL
LIN {X 0,Y 378.026,Z 427.467,A -85,B 0,C 180,E1 -12343.437,E2 -12343.437} C_VEL
LIN {X 0,Y 378.715,Z 416.939,A -85,B 0,C 180,E1 -12344.234,E2 -12344.234} C_VEL
LIN {X 0,Y 379.309,Z 405.668,A -85,B 0,C 180,E1 -12344.828,E2 -12344.828} C_VEL
LIN {X 0,Y 379.774,Z 396.267,A -85,B 0,C 180,E1 -12345.158,E2 -12345.158} C_VEL
LIN {X 0,Y 380.217,Z 361.789,A -85,B 0,C 180,E1 -12345.865,E2 -12345.865} C_VEL
LIN {X 0,Y 380.302,Z 343.401,A -85,B 0,C 180,E1 -12346.231,E2 -12346.231} C_VEL
LIN {X 0,Y 376.751,Z 319.453,A -85,B 0,C 180,E1 -12346.888,E2 -12346.888} C_VEL
LIN {X 0,Y 376.476,Z 317.594,A -85,B 0,C 180,E1 -12346.958,E2 -12346.958} C_VEL
LIN {X 0,Y 377.269,Z 304.849,A -85,B 0,C 180,E1 -12350.158,E2 -12350.158} C_VEL
LIN {X 0,Y 378.029,Z 294.868,A -85,B 0,C 180,E1 -12352.691,E2 -12352.691} C_VEL
LIN {X 0,Y 376.485,Z 285.941,A -85,B 0,C 180,E1 -12355.13,E2 -12355.13} C_VEL
LIN {X 0,Y 375.974,Z 283.465,A -85,B 0,C 180,E1 -12355.857,E2 -12355.857} C_VEL
LIN {X 0,Y 375.913,Z 283.473,A -85,B 0,C 180,E1 -12359.083,E2 -12359.083} C_VEL
LIN {X 0,Y 375.953,Z 283.465,A -85,B 0,C 180,E1 -12361.561,E2 -12361.561} C_VEL
LIN {X 0,Y 375.952,Z 283.469,A -85,B 0,C 180,E1 -12365.415,E2 -12365.415} C_VEL
LIN {X 0,Y 375.967,Z 283.467,A -85,B 0,C 180,E1 -12368.269,E2 -12368.269} C_VEL
LIN {X 0,Y 375.926,Z 283.472,A -85,B 0,C 180,E1 -12371.599,E2 -12371.599} C_VEL
LIN {X 0,Y 375.92,Z 283.473,A -85,B 0,C 180,E1 -12375.268,E2 -12375.268} C_VEL
LIN {X 0,Y 375.926,Z 283.466,A -85,B 0,C 180,E1 -12378.399,E2 -12378.399} C_VEL
LIN {X 0,Y 375.964,Z 283.463,A -85,B 0,C 180,E1 -12381.729,E2 -12381.729} C_VEL
LIN {X 0,Y 375.971,Z 283.465,A -85,B 0,C 180,E1 -12385.332,E2 -12385.332} C_VEL
LIN {X 0,Y 375.948,Z 283.463,A -85,B 0,C 180,E1 -12388.437,E2 -12388.437} C_VEL
LIN {X 0,Y 375.973,Z 283.456,A -85,B 0,C 180,E1 -12392.14,E2 -12392.14} C_VEL
LIN {X 0,Y 375.995,Z 283.46,A -85,B 0,C 180,E1 -12394.538,E2 -12394.538} C_VEL
LIN {X 0,Y 375.946,Z 283.459,A -85,B 0,C 180,E1 -12398.045,E2 -12398.045} C_VEL
LIN {X 0,Y 375.998,Z 283.459,A -85,B 0,C 180,E1 -12401.473,E2 -12401.473} C_VEL
LIN {X 0,Y 376.046,Z 283.447,A -85,B 0,C 180,E1 -12404.832,E2 -12404.832} C_VEL
LIN {X 0,Y 376.039,Z 283.456,A -85,B 0,C 180,E1 -12408.136,E2 -12408.136} C_VEL
LIN {X 0,Y 376.209,Z 283.425,A -85,B 0,C 180,E1 -12411.918,E2 -12411.918} C_VEL
LIN {X 0,Y 376.157,Z 283.441,A -85,B 0,C 180,E1 -12414.64,E2 -12414.64} C_VEL
LIN {X 0,Y 376.339,Z 283.41,A -85,B 0,C 180,E1 -12417.86,E2 -12417.86} C_VEL
LIN {X 0,Y 376.476,Z 283.397,A -85,B 0,C 180,E1 -12420,E2 -12420} C_VEL
LIN {X 0,Y 376.172,Z 283.434,A -85,B 0,C 180,E1 -12423.213,E2 -12423.213} C_VEL
LIN {X 0,Y 376.198,Z 283.432,A -85,B 0,C 180,E1 -12426.464,E2 -12426.464} C_VEL
LIN {X 0,Y 376.107,Z 283.448,A -85,B 0,C 180,E1 -12429.682,E2 -12429.682} C_VEL
LIN {X 0,Y 376.079,Z 283.452,A -85,B 0,C 180,E1 -12433.658,E2 -12433.658} C_VEL
LIN {X 0,Y 376.033,Z 283.457,A -85,B 0,C 180,E1 -12437.607,E2 -12437.607} C_VEL
LIN {X 0,Y 375.969,Z 283.461,A -85,B 0,C 180,E1 -12440.833,E2 -12440.833} C_VEL
LIN {X 0,Y 375.984,Z 283.465,A -85,B 0,C 180,E1 -12444.282,E2 -12444.282} C_VEL
LIN {X 0,Y 376.011,Z 283.457,A -85,B 0,C 180,E1 -12446.653,E2 -12446.653} C_VEL
LIN {X 0,Y 375.968,Z 283.461,A -85,B 0,C 180,E1 -12449.08,E2 -12449.08} C_VEL
LIN {X 0,Y 375.942,Z 283.468,A -85,B 0,C 180,E1 -12452.829,E2 -12452.829} C_VEL
LIN {X 0,Y 375.951,Z 283.463,A -85,B 0,C 180,E1 -12455.416,E2 -12455.416} C_VEL
LIN {X 0,Y 375.971,Z 283.468,A -85,B 0,C 180,E1 -12458.272,E2 -12458.272} C_VEL
LIN {X 0,Y 376.009,Z 283.48,A -85,B 0,C 180,E1 -12461.079,E2 -12461.079} C_VEL
LIN {X 0,Y 377.157,Z 289.423,A -85,B 0,C 180,E1 -12462.764,E2 -12462.764} C_VEL
LIN {X 0,Y 376.858,Z 298.352,A -85,B 0,C 180,E1 -12465.126,E2 -12465.126} C_VEL
LIN {X 0,Y 380.71,Z 318.398,A -85,B 0,C 180,E1 -12465.727,E2 -12465.727} C_VEL
LIN {X 0,Y 379.929,Z 374.818,A -85,B 0,C 180,E1 -12466.851,E2 -12466.851} C_VEL
LIN {X 0,Y 379.6,Z 384.252,A -85,B 0,C 180,E1 -12467.167,E2 -12467.167} C_VEL
LIN {X 0,Y 379.246,Z 394.404,A -85,B 0,C 180,E1 -12467.677,E2 -12467.677} C_VEL
LIN {X 0,Y 378.646,Z 405.229,A -85,B 0,C 180,E1 -12468.43,E2 -12468.43} C_VEL
LIN {X 0,Y 378.017,Z 413.885,A -85,B 0,C 180,E1 -12469.231,E2 -12469.231} C_VEL
LIN {X 0,Y 377.363,Z 422.311,A -85,B 0,C 180,E1 -12470.208,E2 -12470.208} C_VEL
LIN {X 0,Y 376.748,Z 429.288,A -85,B 0,C 180,E1 -12471.197,E2 -12471.197} C_VEL
LIN {X 0,Y 376.233,Z 435.588,A -85,B 0,C 180,E1 -12472.284,E2 -12472.284} C_VEL
LIN {X 0,Y 375.706,Z 441.583,A -85,B 0,C 180,E1 -12473.549,E2 -12473.549} C_VEL
LIN {X 0,Y 375.252,Z 447.322,A -85,B 0,C 180,E1 -12475.074,E2 -12475.074} C_VEL
LIN {X 0,Y 374.889,Z 451.189,A -85,B 0,C 180,E1 -12476.426,E2 -12476.426} C_VEL
LIN {X 0,Y 374.79,Z 453.61,A -85,B 0,C 180,E1 -12477.547,E2 -12477.547} C_VEL
LIN {X 0,Y 374.452,Z 456.494,A -85,B 0,C 180,E1 -12479.553,E2 -12479.553} C_VEL
LIN {X 0,Y 374.325,Z 457.409,A -85,B 0,C 180,E1 -12480.782,E2 -12480.782} C_VEL
LIN {X 0,Y 374.305,Z 457.678,A -85,B 0,C 180,E1 -12482.005,E2 -12482.005} C_VEL
LIN {X 0,Y 374.327,Z 457.285,A -85,B 0,C 180,E1 -12483.219,E2 -12483.219} C_VEL
LIN {X 0,Y 374.421,Z 456.225,A -85,B 0,C 180,E1 -12484.424,E2 -12484.424} C_VEL
LIN {X 0,Y 374.659,Z 453.459,A -85,B 0,C 180,E1 -12486.216,E2 -12486.216} C_VEL
LIN {X 0,Y 374.842,Z 450.828,A -85,B 0,C 180,E1 -12487.397,E2 -12487.397} C_VEL
LIN {X 0,Y 375.133,Z 446.44,A -85,B 0,C 180,E1 -12488.861,E2 -12488.861} C_VEL
LIN {X 0,Y 375.54,Z 440.791,A -85,B 0,C 180,E1 -12490.315,E2 -12490.315} C_VEL
LIN {X 0,Y 375.949,Z 435.197,A -85,B 0,C 180,E1 -12491.471,E2 -12491.471} C_VEL
LIN {X 0,Y 376.442,Z 428.403,A -85,B 0,C 180,E1 -12492.62,E2 -12492.62} C_VEL
LIN {X 0,Y 377.075,Z 420.059,A -85,B 0,C 180,E1 -12493.766,E2 -12493.766} C_VEL
LIN {X 0,Y 377.701,Z 410.756,A -85,B 0,C 180,E1 -12494.763,E2 -12494.763} C_VEL
LIN {X 0,Y 378.318,Z 400.943,A -85,B 0,C 180,E1 -12495.573,E2 -12495.573} C_VEL
LIN {X 0,Y 378.644,Z 392.717,A -85,B 0,C 180,E1 -12496.106,E2 -12496.106} C_VEL
LIN {X 0,Y 378.977,Z 383.265,A -85,B 0,C 180,E1 -12496.563,E2 -12496.563} C_VEL
LIN {X 0,Y 379.229,Z 373.496,A -85,B 0,C 180,E1 -12496.879,E2 -12496.879} C_VEL
LIN {X 0,Y 379.777,Z 317.464,A -85,B 0,C 180,E1 -12497.984,E2 -12497.984} C_VEL
LIN {X 0,Y 376.501,Z 298.657,A -85,B 0,C 180,E1 -12498.493,E2 -12498.493} C_VEL
LIN {X 0,Y 376.913,Z 289.323,A -85,B 0,C 180,E1 -12501.209,E2 -12501.209} C_VEL
LIN {X 0,Y 376.25,Z 283.432,A -85,B 0,C 180,E1 -12503.027,E2 -12503.027} C_VEL
LIN {X 0,Y 376.353,Z 283.42,A -85,B 0,C 180,E1 -12507.86,E2 -12507.86} C_VEL
LIN {X 0,Y 376.489,Z 283.402,A -85,B 0,C 180,E1 -12510,E2 -12510} C_VEL
LIN {X 0,Y 376.186,Z 283.434,A -85,B 0,C 180,E1 -12513.213,E2 -12513.213} C_VEL
LIN {X 0,Y 376.221,Z 283.433,A -85,B 0,C 180,E1 -12516.435,E2 -12516.435} C_VEL
LIN {X 0,Y 376.119,Z 283.443,A -85,B 0,C 180,E1 -12519.691,E2 -12519.691} C_VEL
LIN {X 0,Y 375.407,Z 283.535,A -85,B 0,C 180,E1 -12520.583,E2 -12520.583} C_VEL
LIN {X 0,Y 372.559,Z 283.893,A -85,B 0,C 180,E1 -12522.036,E2 -12522.036} C_VEL
LIN {X 0,Y 370.16,Z 284.196,A -85,B 0,C 180,E1 -12523.21,E2 -12523.21} C_VEL
LIN {X 0,Y 369.109,Z 284.324,A -85,B 0,C 180,E1 -12524.117,E2 -12524.117} C_VEL
LIN {X 0,Y 369.01,Z 284.333,A -85,B 0,C 180,E1 -12524.425,E2 -12524.425} C_VEL
LIN {X 0,Y 368.977,Z 284.332,A -85,B 0,C 180,E1 -12527.756,E2 -12527.756} C_VEL
LIN {X 0,Y 368.91,Z 284.342,A -85,B 0,C 180,E1 -12531.22,E2 -12531.22} C_VEL
LIN {X 0,Y 368.955,Z 284.342,A -85,B 0,C 180,E1 -12534.775,E2 -12534.775} C_VEL
LIN {X 0,Y 368.962,Z 284.337,A -85,B 0,C 180,E1 -12537.203,E2 -12537.203} C_VEL
LIN {X 0,Y 368.917,Z 284.34,A -85,B 0,C 180,E1 -12539.689,E2 -12539.689} C_VEL
LIN {X 0,Y 368.894,Z 284.349,A -85,B 0,C 180,E1 -12543.042,E2 -12543.042} C_VEL
LIN {X 0,Y 368.914,Z 284.34,A -85,B 0,C 180,E1 -12546.196,E2 -12546.196} C_VEL
LIN {X 0,Y 368.9,Z 284.345,A -85,B 0,C 180,E1 -12548.952,E2 -12548.952} C_VEL
LIN {X 0,Y 368.877,Z 284.345,A -85,B 0,C 180,E1 -12552.008,E2 -12552.008} C_VEL
LIN {X 0,Y 368.948,Z 284.339,A -85,B 0,C 180,E1 -12555.186,E2 -12555.186} C_VEL
LIN {X 0,Y 368.94,Z 284.338,A -85,B 0,C 180,E1 -12558.185,E2 -12558.185} C_VEL
LIN {X 0,Y 368.906,Z 284.343,A -85,B 0,C 180,E1 -12561.358,E2 -12561.358} C_VEL
LIN {X 0,Y 368.93,Z 284.338,A -85,B 0,C 180,E1 -12565.146,E2 -12565.146} C_VEL
LIN {X 0,Y 368.922,Z 284.339,A -85,B 0,C 180,E1 -12569.046,E2 -12569.046} C_VEL
LIN {X 0,Y 368.978,Z 284.333,A -85,B 0,C 180,E1 -12571.564,E2 -12571.564} C_VEL
LIN {X 0,Y 368.949,Z 284.335,A -85,B 0,C 180,E1 -12575.224,E2 -12575.224} C_VEL
LIN {X 0,Y 368.928,Z 284.339,A -85,B 0,C 180,E1 -12578.973,E2 -12578.973} C_VEL
LIN {X 0,Y 368.981,Z 284.336,A -85,B 0,C 180,E1 -12582.257,E2 -12582.257} C_VEL
LIN {X 0,Y 369.027,Z 284.328,A -85,B 0,C 180,E1 -12586.227,E2 -12586.227} C_VEL
LIN {X 0,Y 369.057,Z 284.323,A -85,B 0,C 180,E1 -12590.131,E2 -12590.131} C_VEL
LIN {X 0,Y 369.189,Z 284.307,A -85,B 0,C 180,E1 -12593.441,E2 -12593.441} C_VEL
LIN {X 0,Y 369.307,Z 284.291,A -85,B 0,C 180,E1 -12597.819,E2 -12597.819} C_VEL
LIN {X 0,Y 369.446,Z 284.273,A -85,B 0,C 180,E1 -12600,E2 -12600} C_VEL
LIN {X 0,Y 369.305,Z 284.291,A -85,B 0,C 180,E1 -12602.181,E2 -12602.181} C_VEL
LIN {X 0,Y 369.189,Z 284.306,A -85,B 0,C 180,E1 -12606.558,E2 -12606.558} C_VEL
LIN {X 0,Y 369.059,Z 284.324,A -85,B 0,C 180,E1 -12609.868,E2 -12609.868} C_VEL
LIN {X 0,Y 369.027,Z 284.331,A -85,B 0,C 180,E1 -12613.773,E2 -12613.773} C_VEL
LIN {X 0,Y 368.991,Z 284.337,A -85,B 0,C 180,E1 -12617.769,E2 -12617.769} C_VEL
LIN {X 0,Y 368.9,Z 284.342,A -85,B 0,C 180,E1 -12621.221,E2 -12621.221} C_VEL
LIN {X 0,Y 368.945,Z 284.336,A -85,B 0,C 180,E1 -12624.776,E2 -12624.776} C_VEL
LIN {X 0,Y 368.954,Z 284.335,A -85,B 0,C 180,E1 -12627.204,E2 -12627.204} C_VEL
LIN {X 0,Y 368.921,Z 284.339,A -85,B 0,C 180,E1 -12630.954,E2 -12630.954} C_VEL
LIN {X 0,Y 368.921,Z 284.34,A -85,B 0,C 180,E1 -12635.002,E2 -12635.002} C_VEL
LIN {X 0,Y 368.899,Z 284.347,A -85,B 0,C 180,E1 -12638.64,E2 -12638.64} C_VEL
LIN {X 0,Y 368.874,Z 284.346,A -85,B 0,C 180,E1 -12642.01,E2 -12642.01} C_VEL
LIN {X 0,Y 368.877,Z 284.346,A -85,B 0,C 180,E1 -12645.177,E2 -12645.177} C_VEL
LIN {X 0,Y 368.875,Z 284.345,A -85,B 0,C 180,E1 -12648.178,E2 -12648.178} C_VEL
LIN {X 0,Y 368.902,Z 284.344,A -85,B 0,C 180,E1 -12651.361,E2 -12651.361} C_VEL
LIN {X 0,Y 368.932,Z 284.344,A -85,B 0,C 180,E1 -12655.147,E2 -12655.147} C_VEL
LIN {X 0,Y 368.926,Z 284.344,A -85,B 0,C 180,E1 -12659.047,E2 -12659.047} C_VEL
LIN {X 0,Y 368.868,Z 284.35,A -85,B 0,C 180,E1 -12662.79,E2 -12662.79} C_VEL
LIN {X 0,Y 368.923,Z 284.357,A -85,B 0,C 180,E1 -12664.091,E2 -12664.091} C_VEL
LIN {X 0,Y 370.725,Z 293.982,A -85,B 0,C 180,E1 -12666.837,E2 -12666.837} C_VEL
LIN {X 0,Y 370.761,Z 298.557,A -85,B 0,C 180,E1 -12668.075,E2 -12668.075} C_VEL
LIN {X 0,Y 369.627,Z 313.196,A -85,B 0,C 180,E1 -12671.931,E2 -12671.931} C_VEL
LIN {X 0,Y 369.284,Z 318.295,A -85,B 0,C 180,E1 -12673.236,E2 -12673.236} C_VEL
LIN {X 0,Y 372.878,Z 345.721,A -85,B 0,C 180,E1 -12673.941,E2 -12673.941} C_VEL
LIN {X 0,Y 372.204,Z 395.59,A -85,B 0,C 180,E1 -12674.952,E2 -12674.952} C_VEL
LIN {X 0,Y 371.779,Z 405.152,A -85,B 0,C 180,E1 -12675.285,E2 -12675.285} C_VEL
LIN {X 0,Y 371.197,Z 416.695,A -85,B 0,C 180,E1 -12675.891,E2 -12675.891} C_VEL
LIN {X 0,Y 370.59,Z 427.348,A -85,B 0,C 180,E1 -12676.707,E2 -12676.707} C_VEL
LIN {X 0,Y 370.029,Z 435.693,A -85,B 0,C 180,E1 -12677.523,E2 -12677.523} C_VEL
LIN {X 0,Y 369.452,Z 443.591,A -85,B 0,C 180,E1 -12678.479,E2 -12678.479} C_VEL
LIN {X 0,Y 368.866,Z 450.974,A -85,B 0,C 180,E1 -12679.572,E2 -12679.572} C_VEL
LIN {X 0,Y 368.284,Z 458.459,A -85,B 0,C 180,E1 -12680.942,E2 -12680.942} C_VEL
LIN {X 0,Y 367.918,Z 464.316,A -85,B 0,C 180,E1 -12682.316,E2 -12682.316} C_VEL
LIN {X 0,Y 367.577,Z 469.349,A -85,B 0,C 180,E1 -12683.84,E2 -12683.84} C_VEL
LIN {X 0,Y 367.533,Z 472.51,A -85,B 0,C 180,E1 -12685.064,E2 -12685.064} C_VEL
LIN {X 0,Y 367.397,Z 475.564,A -85,B 0,C 180,E1 -12686.71,E2 -12686.71} C_VEL
LIN {X 0,Y 367.364,Z 476.948,A -85,B 0,C 180,E1 -12687.807,E2 -12687.807} C_VEL
LIN {X 0,Y 367.401,Z 477.845,A -85,B 0,C 180,E1 -12688.904,E2 -12688.904} C_VEL
LIN {X 0,Y 367.454,Z 478.163,A -85,B 0,C 180,E1 -12690,E2 -12690} C_VEL
LIN {X 0,Y 367.401,Z 477.945,A -85,B 0,C 180,E1 -12691.096,E2 -12691.096} C_VEL
LIN {X 0,Y 367.361,Z 477.261,A -85,B 0,C 180,E1 -12692.193,E2 -12692.193} C_VEL
LIN {X 0,Y 367.396,Z 476.103,A -85,B 0,C 180,E1 -12693.29,E2 -12693.29} C_VEL
LIN {X 0,Y 367.51,Z 474.426,A -85,B 0,C 180,E1 -12694.387,E2 -12694.387} C_VEL
LIN {X 0,Y 367.611,Z 470.253,A -85,B 0,C 180,E1 -12696.208,E2 -12696.208} C_VEL
LIN {X 0,Y 367.878,Z 467.58,A -85,B 0,C 180,E1 -12697.133,E2 -12697.133} C_VEL
LIN {X 0,Y 368.146,Z 462.555,A -85,B 0,C 180,E1 -12698.508,E2 -12698.508} C_VEL
LIN {X 0,Y 368.704,Z 456.246,A -85,B 0,C 180,E1 -12699.878,E2 -12699.878} C_VEL
LIN {X 0,Y 369.256,Z 450.08,A -85,B 0,C 180,E1 -12700.972,E2 -12700.972} C_VEL
LIN {X 0,Y 369.812,Z 443.612,A -85,B 0,C 180,E1 -12701.927,E2 -12701.927} C_VEL
LIN {X 0,Y 370.473,Z 435.789,A -85,B 0,C 180,E1 -12702.879,E2 -12702.879} C_VEL
LIN {X 0,Y 371.139,Z 427.553,A -85,B 0,C 180,E1 -12703.692,E2 -12703.692} C_VEL
LIN {X 0,Y 371.863,Z 417.108,A -85,B 0,C 180,E1 -12704.502,E2 -12704.502} C_VEL
